(* CODESYS project CANopenExample.project
   Title: CANopen Example

Project tree, tasks and I/O mapping:
  Device : CODESYS Control Win V3 x64, 3S - Smart Software Solutions GmbH, version 3.5.14.0
    application Application
      libraries: Standard, * (System); MemoryUtils, * (3S - Smart Software Solutions GmbH); StringUtils, * (System); CmpLog, * (System); CAA CiA 405, 3.5.14.0 (CAA Technical Workgroup)
      task MainTask (cyclic, interval t#20ms, priority 1) calls CANopenManagerExamples, CANopenLocalDeviceExamples, CANbusExamples
      CANbus Examples/
        program CANbusExamples [ST]
        Change CANbus settings (Reconfigure)/
          program ChangeBaudrate [ST]
          program EnableDisableCANbus [ST]
        Query CANbus/
          function GetCANbus [ST]
      CANopen Master Examples/
        program CANopenManagerExamples [ST]
        CiA405/
          Diagnosis/
            EMCY/
              program ReceiveEMCYFromAllDevicesExample [ST]
              program ReceiveEMCYFromOneDeviceExample [ST]
            State/
              program GetCANopenKernelStateExample [ST]
              program GetStateExample [ST]
          Network management/
            program GetCANopenManagerNodeIDExample [ST]
            program NMT_Example [ST]
          SDO access/
            Block and Segmented/
              program SegmentedAndBlockReadExample [ST]
              program SegmentedAndBlockWriteExample [ST]
            Expedited (<= 4byte)/
              program ExpeditedReadExample [ST]
              program ExpeditedWriteExample [ST]
        Stack API/
          program CANopenManagerAPI [ST]
          program CANopenRemoteDeviceAPI [ST]
          Events/
            function block CANopenManagerEventHandler [ST]: EventCallback
      CANopen Slave Examples/
        program CANopenLocalDeviceExamples [ST]
        Diagnosis/
          function GetLocalDeviceInfoExample [ST]
        Network management/
          program ChangeNodeIDExample [ST]
          program NMTExample [ST]
          data type NMT_Command
        Object Dictionary Access/
          Event Handler/
            function block ObjectDictionaryEventHandler [ST]: OnObjectChanged, OnReadObject, OnWriteObject
            function TO_HEXSTRING [ST]
          Read Object/
            program ReadObjectExample1 [ST]
            program ReadObjectExample2 [ST]
          Traverse object dictionary/
            program CountObjects [ST]
            program GetPDOInfo [ST]
          Write Object/
            program WriteObjectExample1 [ST]
            program WriteObjectExample2 [ST]
      license
    CANbus : CANbus, 3S - Smart Software Solutions GmbH, version 3.5.12.0
        settings: Baudrate = 1000 kbit/s
      CANopen_Manager : CANopen_Manager, 3S - Smart Software Solutions GmbH, version 3.5.10.0
          settings: ConfigVersion = 50659584
        CANopenRemoteDevice : CANopenDeviceExample, 3S - Smart Software Solutions GmbH, order no. 0, version Revision=16#00000004, FileVersion=1.0
            settings: NODEIDSAVED = 1; SDO Timeout = 1000000; EXPERTSETTINGS = FALSE; Heartbeat-Producer Time = 200; PDO 16#1400.COBID = 16#00000201; Process by CANopenManager = TRUE; PDO 16#1800.COBID = 16#00000181; Process by CANopenManager = TRUE; Heartbeat-Consuming1.Heartbeat-Time = 300 ms; DigOutput8.Subindex = 16#01; DigOutput8.Subindex = 16#02; DigOutput8.Subindex = 16#03; DigOutput8.Subindex = 16#04; DigOutput8.Subindex = 16#05; DigOutput8.Subindex = 16#06; DigOutput8.Subindex = 16#07; DigOutput8.Subindex = 16#08; DigInput8.Subindex = 16#01; DigInput8.Subindex = 16#02; DigInput8.Subindex = 16#03; DigInput8.Subindex = 16#04; DigInput8.Subindex = 16#05; DigInput8.Subindex = 16#06; DigInput8.Subindex = 16#07; DigInput8.Subindex = 16#08; SDO List.Set Guardtime.Index = 16#100C; SDO List.Set Guardtime.Subindex = 16#00; SDO List.Set Guardtime.Value = 16#00000000; SDO List.Set Guardtime.Size = 16; SDO List.Set Guardtime.AbortIfError = FALSE; SDO List.Set Guardtime.JumpToLine = FALSE; SDO List.Set Guardtime.Line = 0; SDO List.Set Lifetime.Index = 16#100D; SDO List.Set Lifetime.Subindex = 16#00; SDO List.Set Lifetime.Value = 16#00000000; SDO List.Set Lifetime.Size = 8; SDO List.Set Lifetime.AbortIfError = FALSE; SDO List.Set Lifetime.JumpToLine = FALSE; SDO List.Set Lifetime.Line = 0; SDO List.Disable Emcy CobID.Index = 16#1014;
              SDO List.Disable Emcy CobID.Subindex = 16#00; SDO List.Disable Emcy CobID.Value = 16#80000081; SDO List.Disable Emcy CobID.Size = 32; SDO List.Disable Emcy CobID.AbortIfError = FALSE; SDO List.Disable Emcy CobID.JumpToLine = FALSE; SDO List.Disable Emcy CobID.Line = 0; SDO List.Set Emcy CobID.Index = 16#1014; SDO List.Set Emcy CobID.Subindex = 16#00; SDO List.Set Emcy CobID.Value = 16#00000081; SDO List.Set Emcy CobID.Size = 32; SDO List.Set Emcy CobID.AbortIfError = FALSE; SDO List.Set Emcy CobID.JumpToLine = FALSE; SDO List.Set Emcy CobID.Line = 0; SDO List.Set Heartbeat Consumer.Index = 16#1016; SDO List.Set Heartbeat Consumer.Subindex = 16#01; SDO List.Set Heartbeat Consumer.Value = 16#007F012C; SDO List.Set Heartbeat Consumer.Size = 32; SDO List.Set Heartbeat Consumer.AbortIfError = FALSE; SDO List.Set Heartbeat Consumer.JumpToLine = FALSE; SDO List.Set Heartbeat Consumer.Line = 0; SDO List.Set Heartbeat Producer.Index = 16#1017; SDO List.Set Heartbeat Producer.Subindex = 16#00; SDO List.Set Heartbeat Producer.Value = 16#000000C8; SDO List.Set Heartbeat Producer.Size = 16; SDO List.Set Heartbeat Producer.AbortIfError = FALSE; SDO List.Set Heartbeat Producer.JumpToLine = FALSE; SDO List.Set Heartbeat Producer.Line = 0; SDO List.Disable PDO.Index = 16#1400; SDO List.Disable PDO.Subindex = 16#01; SDO List.Disable PDO.Value = 16#80000201; SDO List.Disable PDO.Size = 32; SDO List.Disable PDO.AbortIfError = FALSE; SDO List.Disable PDO.JumpToLine = FALSE; SDO List.Disable PDO.Line = 0; SDO List.Set transmission type.Index = 16#1400; SDO List.Set transmission type.Subindex = 16#02; SDO List.Set transmission type.Value = 16#FF; SDO List.Set transmission type.Size = 8; SDO List.Set transmission type.AbortIfError = FALSE; SDO List.Set transmission type.JumpToLine = FALSE;
              SDO List.Set transmission type.Line = 0; SDO List.Set and enable COB-ID.Index = 16#1400; SDO List.Set and enable COB-ID.Subindex = 16#01; SDO List.Set and enable COB-ID.Value = 16#00000201; SDO List.Set and enable COB-ID.Size = 32; SDO List.Set and enable COB-ID.AbortIfError = FALSE; SDO List.Set and enable COB-ID.JumpToLine = FALSE; SDO List.Set and enable COB-ID.Line = 0; SDO List.Disable PDO.Index = 16#1800; SDO List.Disable PDO.Subindex = 16#01; SDO List.Disable PDO.Value = 16#80000181; SDO List.Disable PDO.Size = 32; SDO List.Disable PDO.AbortIfError = FALSE; SDO List.Disable PDO.JumpToLine = FALSE; SDO List.Disable PDO.Line = 0; SDO List.Set transmission type.Index = 16#1800; SDO List.Set transmission type.Subindex = 16#02; SDO List.Set transmission type.Value = 16#FF; SDO List.Set transmission type.Size = 8; SDO List.Set transmission type.AbortIfError = FALSE; SDO List.Set transmission type.JumpToLine = FALSE; SDO List.Set transmission type.Line = 0; SDO List.Set inhibit time.Index = 16#1800; SDO List.Set inhibit time.Subindex = 16#03; SDO List.Set inhibit time.Value = 16#0000; SDO List.Set inhibit time.Size = 16; SDO List.Set inhibit time.AbortIfError = FALSE; SDO List.Set inhibit time.JumpToLine = FALSE; SDO List.Set inhibit time.Line = 0; SDO List.Set event time.Index = 16#1800; SDO List.Set event time.Subindex = 16#05; SDO List.Set event time.Value = 16#0000; SDO List.Set event time.Size = 16; SDO List.Set event time.AbortIfError = FALSE; SDO List.Set event time.JumpToLine = FALSE; SDO List.Set event time.Line = 0; SDO List.Set and enable COB-ID.Index = 16#1800; SDO List.Set and enable COB-ID.Subindex = 16#01; SDO List.Set and enable COB-ID.Value = 16#00000181; SDO List.Set and enable COB-ID.Size = 32;
              SDO List.Set and enable COB-ID.AbortIfError = FALSE; SDO List.Set and enable COB-ID.JumpToLine = FALSE; SDO List.Set and enable COB-ID.Line = 0; ConfigVersion = 50659584
            unmapped channels: DigOutput8, DigOutput8, DigOutput8, DigOutput8, DigOutput8, DigOutput8, DigOutput8, DigOutput8, DigInput8, DigInput8, DigInput8, DigInput8, DigInput8, DigInput8, DigInput8, DigInput8
    CANbus_1 : CANbus, 3S - Smart Software Solutions GmbH, version 3.5.12.0
        settings: Baudrate = 1000 kbit/s
      CANopenLocalDevice : CANopen Device, 3S - Smart Software Solutions GmbH, version 3.5.13.0
          settings: Product Name = 'CANopenDeviceExample'; OD_ObjectCount = 16#0015; Objects.Objects = (wIndex := 16#1000, bySubCnt := 16#1); Objects.Objects = (wIndex := 16#1001, bySubCnt := 16#1); Objects.Objects = (wIndex := 16#1003, bySubCnt := 16#04); Objects.Objects = (wIndex := 16#1005, bySubCnt := 16#1); Objects.Objects = (wIndex := 16#1006, bySubCnt := 16#1); Objects.Objects = (wIndex := 16#1008, bySubCnt := 16#1); Objects.Objects = (wIndex := 16#100C, bySubCnt := 16#1); Objects.Objects = (wIndex := 16#100D, bySubCnt := 16#1); Objects.Objects = (wIndex := 16#1014, bySubCnt := 16#1); Objects.Objects = (wIndex := 16#1016, bySubCnt := 16#02); Objects.Objects = (wIndex := 16#1017, bySubCnt := 16#1); Objects.Objects = (wIndex := 16#1018, bySubCnt := 16#04); Objects.Objects = (wIndex := 16#1200, bySubCnt := 16#03); Objects.Objects = (wIndex := 16#1400, bySubCnt := 16#03); Objects.Objects = (wIndex := 16#1600, bySubCnt := 16#09); Objects.Objects = (wIndex := 16#1800, bySubCnt := 16#06); Objects.Objects = (wIndex := 16#1A00, bySubCnt := 16#09); Objects.Objects = (wIndex := 16#3000, bySubCnt := 16#1); Objects.Objects = (wIndex := 16#6000, bySubCnt := 16#09); Objects.Objects = (wIndex := 16#6200, bySubCnt := 16#09); Objects.Objects = (wIndex := 16#6412, bySubCnt := 16#02); SubObjects.SubObjects = (eObjProperties := 16#0001, eDataType := 16#05, udiSize := 16#00000001, xwData := 0, xwDefault := 0, bySubIdx := 16#00); SubObjects.SubObjects = (eObjProperties := 16#0003, eDataType := 16#05, udiSize := 16#00000001, xwData := 0, xwDefault := 0, bySubIdx := 16#00); SubObjects.SubObjects = (eObjProperties := 16#0001, eDataType := 16#07, udiSize := 16#00000004, xwData := 0, xwDefault := 0, bySubIdx := 16#01); SubObjects.SubObjects = (eObjProperties := 16#0001, eDataType := 16#07, udiSize := 16#00000004, xwData := 0, xwDefault := 0, bySubIdx := 16#02); SubObjects.SubObjects = (eObjProperties := 16#0001, eDataType := 16#07, udiSize := 16#00000004, xwData := 0, xwDefault := 0, bySubIdx := 16#03); SubObjects.SubObjects = (eObjProperties := 16#0003, eDataType := 16#07, udiSize := 16#00000004, xwData := 0, xwDefault := 0, bySubIdx := 16#00); SubObjects.SubObjects = (eObjProperties := 16#0001, eDataType := 16#09, udiSize := 20, xwData := 0, xwDefault := 0, bySubIdx := 16#00); SubObjects.SubObjects = (eObjProperties := 16#0003, eDataType := 16#06, udiSize := 16#00000002, xwData := 0, xwDefault := 0, bySubIdx := 16#00); SubObjects.SubObjects = (eObjProperties := 16#0003, eDataType := 16#05, udiSize := 16#00000001, xwData := 0, xwDefault := 0, bySubIdx := 16#00); SubObjects.SubObjects = (eObjProperties := 16#0001, eDataType := 16#05, udiSize := 16#00000001, xwData := 0, xwDefault := 1, bySubIdx := 16#00); SubObjects.SubObjects = (eObjProperties := 16#0003, eDataType := 16#07, udiSize := 16#00000004, xwData := 0, xwDefault := 0, bySubIdx := 16#01); SubObjects.SubObjects = (eObjProperties := 16#0003, eDataType := 16#06, udiSize := 16#00000002, xwData := 0, xwDefault := 0, bySubIdx := 16#00); SubObjects.SubObjects = (eObjProperties := 16#0001, eDataType := 16#05, udiSize := 16#00000001, xwData := 0, xwDefault := 3, bySubIdx := 16#00); SubObjects.SubObjects = (eObjProperties := 16#0001, eDataType := 16#07, udiSize := 16#00000004, xwData := 0, xwDefault := 4, bySubIdx := 16#03); SubObjects.SubObjects = (eObjProperties := 16#0001, eDataType := 16#05, udiSize := 16#00000001, xwData := 0, xwDefault := 2, bySubIdx := 16#00); SubObjects.SubObjects = (eObjProperties := 16#0001, eDataType := 16#05, udiSize := 16#00000001, xwData := 0, xwDefault := 2, bySubIdx := 16#00); SubObjects.SubObjects = (eObjProperties := 16#0001, eDataType := 16#05, udiSize := 16#00000001, xwData := 0, xwDefault := 8, bySubIdx := 16#00);
            SubObjects.SubObjects = (eObjProperties := 16#0001, eDataType := 16#05, udiSize := 16#00000001, xwData := 0, xwDefault := 5, bySubIdx := 16#00); SubObjects.SubObjects = (eObjProperties := 16#0003, eDataType := 16#06, udiSize := 16#00000002, xwData := 0, xwDefault := 0, bySubIdx := 16#03); SubObjects.SubObjects = (eObjProperties := 16#0003, eDataType := 16#05, udiSize := 16#00000001, xwData := 0, xwDefault := 0, bySubIdx := 16#04); SubObjects.SubObjects = (eObjProperties := 16#0003, eDataType := 16#06, udiSize := 16#00000002, xwData := 0, xwDefault := 0, bySubIdx := 16#05); SubObjects.SubObjects = (eObjProperties := 16#0001, eDataType := 16#05, udiSize := 16#00000001, xwData := 0, xwDefault := 8, bySubIdx := 16#00); SubObjects.SubObjects = (eObjProperties := 16#0001, eDataType := 16#05, udiSize := 16#00000001, xwData := 0, xwDefault := 8, bySubIdx := 16#00); SubObjects.SubObjects = (eObjProperties := 16#0001, eDataType := 16#05, udiSize := 16#00000001, xwData := 0, xwDefault := 0, bySubIdx := 16#01); SubObjects.SubObjects = (eObjProperties := 16#0001, eDataType := 16#05, udiSize := 16#00000001, xwData := 0, xwDefault := 0, bySubIdx := 16#02); SubObjects.SubObjects = (eObjProperties := 16#0001, eDataType := 16#05, udiSize := 16#00000001, xwData := 0, xwDefault := 0, bySubIdx := 16#03); SubObjects.SubObjects = (eObjProperties := 16#0001, eDataType := 16#05, udiSize := 16#00000001, xwData := 0, xwDefault := 0, bySubIdx := 16#04); SubObjects.SubObjects = (eObjProperties := 16#0001, eDataType := 16#05, udiSize := 16#00000001, xwData := 0, xwDefault := 0, bySubIdx := 16#05); SubObjects.SubObjects = (eObjProperties := 16#0001, eDataType := 16#05, udiSize := 16#00000001, xwData := 0, xwDefault := 0, bySubIdx := 16#06); SubObjects.SubObjects = (eObjProperties := 16#0001, eDataType := 16#05, udiSize := 16#00000001, xwData := 0, xwDefault := 0, bySubIdx := 16#07); SubObjects.SubObjects = (eObjProperties := 16#0001, eDataType := 16#05, udiSize := 16#00000001, xwData := 0, xwDefault := 0, bySubIdx := 16#08); SubObjects.SubObjects = (eObjProperties := 16#0001, eDataType := 16#05, udiSize := 16#00000001, xwData := 0, xwDefault := 8, bySubIdx := 16#00); SubObjects.SubObjects = (eObjProperties := 16#0003, eDataType := 16#05, udiSize := 16#00000001, xwData := 0, xwDefault := 0, bySubIdx := 16#01); SubObjects.SubObjects = (eObjProperties := 16#0003, eDataType := 16#05, udiSize := 16#00000001, xwData := 0, xwDefault := 0, bySubIdx := 16#02); SubObjects.SubObjects = (eObjProperties := 16#0003, eDataType := 16#05, udiSize := 16#00000001, xwData := 0, xwDefault := 0, bySubIdx := 16#03); SubObjects.SubObjects = (eObjProperties := 16#0003, eDataType := 16#05, udiSize := 16#00000001, xwData := 0, xwDefault := 0, bySubIdx := 16#04); SubObjects.SubObjects = (eObjProperties := 16#0003, eDataType := 16#05, udiSize := 16#00000001, xwData := 0, xwDefault := 0, bySubIdx := 16#05); SubObjects.SubObjects = (eObjProperties := 16#0003, eDataType := 16#05, udiSize := 16#00000001, xwData := 0, xwDefault := 0, bySubIdx := 16#06); SubObjects.SubObjects = (eObjProperties := 16#0003, eDataType := 16#05, udiSize := 16#00000001, xwData := 0, xwDefault := 0, bySubIdx := 16#07); SubObjects.SubObjects = (eObjProperties := 16#0003, eDataType := 16#05, udiSize := 16#00000001, xwData := 0, xwDefault := 0, bySubIdx := 16#08); SubObjects.SubObjects = (eObjProperties := 16#0001, eDataType := 16#05, udiSize := 16#00000001, xwData := 0, xwDefault := 1, bySubIdx := 16#00); SubObjects.SubObjects = (eObjProperties := 16#0003, eDataType := 16#04, udiSize := 16#00000004, xwData := 0, xwDefault := 0, bySubIdx := 16#01); ObjectsOfflineInfo.Predefined Error Field.Index = 16#00001003; ObjectsOfflineInfo.Predefined Error Field.ObjectOwner = 16#00; ObjectsOfflineInfo.Predefined Error Field.ObjectType = 16#00000008; ObjectsOfflineInfo.Predefined Error Field.ObjectFlags = 16#00000000; ObjectsOfflineInfo.Consumer Heartbeat Time.Index = 16#00001016; ObjectsOfflineInfo.Consumer Heartbeat Time.ObjectOwner = 16#00; ObjectsOfflineInfo.Consumer Heartbeat Time.ObjectType = 16#00000008; ObjectsOfflineInfo.Consumer Heartbeat Time.ObjectFlags = 16#00000000; ObjectsOfflineInfo.Identity Object.Index = 16#00001018; ObjectsOfflineInfo.Identity Object.ObjectOwner = 16#00; ObjectsOfflineInfo.Identity Object.ObjectType = 16#00000009; ObjectsOfflineInfo.Identity Object.ObjectFlags = 16#00000000; ObjectsOfflineInfo.ServerSdoParameter.Index = 16#00001200; ObjectsOfflineInfo.ServerSdoParameter.ObjectOwner = 16#00; ObjectsOfflineInfo.ServerSdoParameter.ObjectType = 16#00000009;
            ObjectsOfflineInfo.ServerSdoParameter.ObjectFlags = 16#00000000; ObjectsOfflineInfo.RPDO communication parameter.Index = 16#00001400; ObjectsOfflineInfo.RPDO communication parameter.ObjectOwner = 16#03; ObjectsOfflineInfo.RPDO communication parameter.ObjectType = 16#00000009; ObjectsOfflineInfo.RPDO communication parameter.ObjectFlags = 16#00000000; ObjectsOfflineInfo.RPDO mapping parameter.Index = 16#00001600; ObjectsOfflineInfo.RPDO mapping parameter.ObjectOwner = 16#03; ObjectsOfflineInfo.RPDO mapping parameter.ObjectType = 16#00000009; ObjectsOfflineInfo.RPDO mapping parameter.ObjectFlags = 16#00000000; ObjectsOfflineInfo.TPDO communication parameter.Index = 16#00001800; ObjectsOfflineInfo.TPDO communication parameter.ObjectOwner = 16#03; ObjectsOfflineInfo.TPDO communication parameter.ObjectType = 16#00000009; ObjectsOfflineInfo.TPDO communication parameter.ObjectFlags = 16#00000000; ObjectsOfflineInfo.TPDO mapping parameter.Index = 16#00001A00; ObjectsOfflineInfo.TPDO mapping parameter.ObjectOwner = 16#03; ObjectsOfflineInfo.TPDO mapping parameter.ObjectType = 16#00000009; ObjectsOfflineInfo.TPDO mapping parameter.ObjectFlags = 16#00000000; ObjectsOfflineInfo.Read Input 8 Bit.Index = 16#00006000; ObjectsOfflineInfo.Read Input 8 Bit.ObjectOwner = 16#03; ObjectsOfflineInfo.Read Input 8 Bit.ObjectType = 16#00000008; ObjectsOfflineInfo.Read Input 8 Bit.ObjectFlags = 16#00000000; ObjectsOfflineInfo.Write Output 8 Bit.Index = 16#00006200; ObjectsOfflineInfo.Write Output 8 Bit.ObjectOwner = 16#03; ObjectsOfflineInfo.Write Output 8 Bit.ObjectType = 16#00000008; ObjectsOfflineInfo.Write Output 8 Bit.ObjectFlags = 16#00000000; ObjectsOfflineInfo.Write Analogue Output 32 Bit.Index = 16#00006412; ObjectsOfflineInfo.Write Analogue Output 32 Bit.ObjectOwner = 16#03; ObjectsOfflineInfo.Write Analogue Output 32 Bit.ObjectType = 16#00000008; ObjectsOfflineInfo.Write Analogue Output 32 Bit.ObjectFlags = 16#00000000; SubObjectsOfflineInfo.Device Type.Index = 16#00001000; SubObjectsOfflineInfo.Device Type.SubIndex = 16#00; SubObjectsOfflineInfo.Device Type.PDOMapping = FALSE; SubObjectsOfflineInfo.Device Type.ObjectOwner = 16#00; SubObjectsOfflineInfo.Device Type.ObjectType = 16#00000007; SubObjectsOfflineInfo.Device Type.MinValue = ''; SubObjectsOfflineInfo.Device Type.MaxValue = ''; SubObjectsOfflineInfo.Device Type.AccessType = 'ro'; SubObjectsOfflineInfo.Device Type.IEC Variable = ''; SubObjectsOfflineInfo.Device Type.DefaultValue = '0x191'; SubObjectsOfflineInfo.Device Type.ObjectFlags = 16#00000000;
            SubObjectsOfflineInfo.Error Register.Index = 16#00001001; SubObjectsOfflineInfo.Error Register.SubIndex = 16#00; SubObjectsOfflineInfo.Error Register.PDOMapping = FALSE; SubObjectsOfflineInfo.Error Register.ObjectOwner = 16#00; SubObjectsOfflineInfo.Error Register.ObjectType = 16#00000007; SubObjectsOfflineInfo.Error Register.MinValue = ''; SubObjectsOfflineInfo.Error Register.MaxValue = ''; SubObjectsOfflineInfo.Error Register.AccessType = 'ro'; SubObjectsOfflineInfo.Error Register.IEC Variable = ''; SubObjectsOfflineInfo.Error Register.DefaultValue = '0x0'; SubObjectsOfflineInfo.Error Register.ObjectFlags = 16#00000000; SubObjectsOfflineInfo.Number of Errors.Index = 16#00001003; SubObjectsOfflineInfo.Number of Errors.SubIndex = 16#00; SubObjectsOfflineInfo.Number of Errors.PDOMapping = FALSE; SubObjectsOfflineInfo.Number of Errors.ObjectOwner = 16#00; SubObjectsOfflineInfo.Number of Errors.ObjectType = 16#00000007; SubObjectsOfflineInfo.Number of Errors.MinValue = ''; SubObjectsOfflineInfo.Number of Errors.MaxValue = ''; SubObjectsOfflineInfo.Number of Errors.AccessType = 'rw'; SubObjectsOfflineInfo.Number of Errors.IEC Variable = ''; SubObjectsOfflineInfo.Number of Errors.DefaultValue = '0'; SubObjectsOfflineInfo.Number of Errors.ObjectFlags = 16#00000000; SubObjectsOfflineInfo.Standard Error Field.Index = 16#00001003; SubObjectsOfflineInfo.Standard Error Field.SubIndex = 16#01; SubObjectsOfflineInfo.Standard Error Field.PDOMapping = FALSE; SubObjectsOfflineInfo.Standard Error Field.ObjectOwner = 16#00; SubObjectsOfflineInfo.Standard Error Field.ObjectType = 16#00000007; SubObjectsOfflineInfo.Standard Error Field.MinValue = ''; SubObjectsOfflineInfo.Standard Error Field.MaxValue = ''; SubObjectsOfflineInfo.Standard Error Field.AccessType = 'ro'; SubObjectsOfflineInfo.Standard Error Field.IEC Variable = ''; SubObjectsOfflineInfo.Standard Error Field.DefaultValue = ''; SubObjectsOfflineInfo.Standard Error Field.ObjectFlags = 16#00000000; SubObjectsOfflineInfo.Standard Error Field 2.Index = 16#00001003; SubObjectsOfflineInfo.Standard Error Field 2.SubIndex = 16#02; SubObjectsOfflineInfo.Standard Error Field 2.PDOMapping = FALSE; SubObjectsOfflineInfo.Standard Error Field 2.ObjectOwner = 16#00; SubObjectsOfflineInfo.Standard Error Field 2.ObjectType = 16#00000007; SubObjectsOfflineInfo.Standard Error Field 2.MinValue = ''; SubObjectsOfflineInfo.Standard Error Field 2.MaxValue = '';
            SubObjectsOfflineInfo.Standard Error Field 2.AccessType = 'ro'; SubObjectsOfflineInfo.Standard Error Field 2.IEC Variable = ''; SubObjectsOfflineInfo.Standard Error Field 2.DefaultValue = ''; SubObjectsOfflineInfo.Standard Error Field 2.ObjectFlags = 16#00000000; SubObjectsOfflineInfo.Standard Error Field 3.Index = 16#00001003; SubObjectsOfflineInfo.Standard Error Field 3.SubIndex = 16#03; SubObjectsOfflineInfo.Standard Error Field 3.PDOMapping = FALSE; SubObjectsOfflineInfo.Standard Error Field 3.ObjectOwner = 16#00; SubObjectsOfflineInfo.Standard Error Field 3.ObjectType = 16#00000007; SubObjectsOfflineInfo.Standard Error Field 3.MinValue = ''; SubObjectsOfflineInfo.Standard Error Field 3.MaxValue = ''; SubObjectsOfflineInfo.Standard Error Field 3.AccessType = 'ro'; SubObjectsOfflineInfo.Standard Error Field 3.IEC Variable = ''; SubObjectsOfflineInfo.Standard Error Field 3.DefaultValue = ''; SubObjectsOfflineInfo.Standard Error Field 3.ObjectFlags = 16#00000000; SubObjectsOfflineInfo.Sync COB-ID.Index = 16#00001005; SubObjectsOfflineInfo.Sync COB-ID.SubIndex = 16#00; SubObjectsOfflineInfo.Sync COB-ID.PDOMapping = FALSE; SubObjectsOfflineInfo.Sync COB-ID.ObjectOwner = 16#00; SubObjectsOfflineInfo.Sync COB-ID.ObjectType = 16#00000007; SubObjectsOfflineInfo.Sync COB-ID.MinValue = ''; SubObjectsOfflineInfo.Sync COB-ID.MaxValue = ''; SubObjectsOfflineInfo.Sync COB-ID.AccessType = 'rw'; SubObjectsOfflineInfo.Sync COB-ID.IEC Variable = ''; SubObjectsOfflineInfo.Sync COB-ID.DefaultValue = '0x80'; SubObjectsOfflineInfo.Sync COB-ID.ObjectFlags = 16#00000000; SubObjectsOfflineInfo.Communication Cycle Period.Index = 16#00001006; SubObjectsOfflineInfo.Communication Cycle Period.SubIndex = 16#00; SubObjectsOfflineInfo.Communication Cycle Period.PDOMapping = FALSE; SubObjectsOfflineInfo.Communication Cycle Period.ObjectOwner = 16#00; SubObjectsOfflineInfo.Communication Cycle Period.ObjectType = 16#00000007; SubObjectsOfflineInfo.Communication Cycle Period.MinValue = ''; SubObjectsOfflineInfo.Communication Cycle Period.MaxValue = ''; SubObjectsOfflineInfo.Communication Cycle Period.AccessType = 'rw'; SubObjectsOfflineInfo.Communication Cycle Period.IEC Variable = ''; SubObjectsOfflineInfo.Communication Cycle Period.DefaultValue = '0x0'; SubObjectsOfflineInfo.Communication Cycle Period.ObjectFlags = 16#00000000; SubObjectsOfflineInfo.Manufacturer device name.Index = 16#00001008; SubObjectsOfflineInfo.Manufacturer device name.SubIndex = 16#00; SubObjectsOfflineInfo.Manufacturer device name.PDOMapping = FALSE;
            SubObjectsOfflineInfo.Manufacturer device name.ObjectOwner = 16#03; SubObjectsOfflineInfo.Manufacturer device name.ObjectType = 16#00000007; SubObjectsOfflineInfo.Manufacturer device name.MinValue = ''; SubObjectsOfflineInfo.Manufacturer device name.MaxValue = ''; SubObjectsOfflineInfo.Manufacturer device name.AccessType = 'const'; SubObjectsOfflineInfo.Manufacturer device name.IEC Variable = ''; SubObjectsOfflineInfo.Manufacturer device name.DefaultValue = 'CANopenDeviceExample'; SubObjectsOfflineInfo.Manufacturer device name.ObjectFlags = 16#00000000; SubObjectsOfflineInfo.Guard Time.Index = 16#0000100C; SubObjectsOfflineInfo.Guard Time.SubIndex = 16#00; SubObjectsOfflineInfo.Guard Time.PDOMapping = FALSE; SubObjectsOfflineInfo.Guard Time.ObjectOwner = 16#00; SubObjectsOfflineInfo.Guard Time.ObjectType = 16#00000007; SubObjectsOfflineInfo.Guard Time.MinValue = ''; SubObjectsOfflineInfo.Guard Time.MaxValue = ''; SubObjectsOfflineInfo.Guard Time.AccessType = 'rw'; SubObjectsOfflineInfo.Guard Time.IEC Variable = ''; SubObjectsOfflineInfo.Guard Time.DefaultValue = '0x0'; SubObjectsOfflineInfo.Guard Time.ObjectFlags = 16#00000000; SubObjectsOfflineInfo.Life Time Factor.Index = 16#0000100D; SubObjectsOfflineInfo.Life Time Factor.SubIndex = 16#00; SubObjectsOfflineInfo.Life Time Factor.PDOMapping = FALSE; SubObjectsOfflineInfo.Life Time Factor.ObjectOwner = 16#00; SubObjectsOfflineInfo.Life Time Factor.ObjectType = 16#00000007; SubObjectsOfflineInfo.Life Time Factor.MinValue = ''; SubObjectsOfflineInfo.Life Time Factor.MaxValue = ''; SubObjectsOfflineInfo.Life Time Factor.AccessType = 'rw'; SubObjectsOfflineInfo.Life Time Factor.IEC Variable = ''; SubObjectsOfflineInfo.Life Time Factor.DefaultValue = '0'; SubObjectsOfflineInfo.Life Time Factor.ObjectFlags = 16#00000000; SubObjectsOfflineInfo.COB-ID EMCY.Index = 16#00001014; SubObjectsOfflineInfo.COB-ID EMCY.SubIndex = 16#00; SubObjectsOfflineInfo.COB-ID EMCY.PDOMapping = FALSE; SubObjectsOfflineInfo.COB-ID EMCY.ObjectOwner = 16#00; SubObjectsOfflineInfo.COB-ID EMCY.ObjectType = 16#00000007; SubObjectsOfflineInfo.COB-ID EMCY.MinValue = ''; SubObjectsOfflineInfo.COB-ID EMCY.MaxValue = ''; SubObjectsOfflineInfo.COB-ID EMCY.AccessType = 'rw'; SubObjectsOfflineInfo.COB-ID EMCY.IEC Variable = ''; SubObjectsOfflineInfo.COB-ID EMCY.DefaultValue = '$$NODEID+0x80';
            SubObjectsOfflineInfo.COB-ID EMCY.ObjectFlags = 16#00000000; SubObjectsOfflineInfo.Number of Entries.Index = 16#00001016; SubObjectsOfflineInfo.Number of Entries.SubIndex = 16#00; SubObjectsOfflineInfo.Number of Entries.PDOMapping = FALSE; SubObjectsOfflineInfo.Number of Entries.ObjectOwner = 16#00; SubObjectsOfflineInfo.Number of Entries.ObjectType = 16#00000007; SubObjectsOfflineInfo.Number of Entries.MinValue = ''; SubObjectsOfflineInfo.Number of Entries.MaxValue = ''; SubObjectsOfflineInfo.Number of Entries.AccessType = 'ro'; SubObjectsOfflineInfo.Number of Entries.IEC Variable = ''; SubObjectsOfflineInfo.Number of Entries.DefaultValue = '0x1'; SubObjectsOfflineInfo.Number of Entries.ObjectFlags = 16#00000000; SubObjectsOfflineInfo.Consumer Heartbeat Time.Index = 16#00001016; SubObjectsOfflineInfo.Consumer Heartbeat Time.SubIndex = 16#01; SubObjectsOfflineInfo.Consumer Heartbeat Time.PDOMapping = FALSE; SubObjectsOfflineInfo.Consumer Heartbeat Time.ObjectOwner = 16#00; SubObjectsOfflineInfo.Consumer Heartbeat Time.ObjectType = 16#00000007; SubObjectsOfflineInfo.Consumer Heartbeat Time.MinValue = ''; SubObjectsOfflineInfo.Consumer Heartbeat Time.MaxValue = ''; SubObjectsOfflineInfo.Consumer Heartbeat Time.AccessType = 'rw'; SubObjectsOfflineInfo.Consumer Heartbeat Time.IEC Variable = ''; SubObjectsOfflineInfo.Consumer Heartbeat Time.DefaultValue = '0x0'; SubObjectsOfflineInfo.Consumer Heartbeat Time.ObjectFlags = 16#00000000; SubObjectsOfflineInfo.Producer Heartbeat Time.Index = 16#00001017; SubObjectsOfflineInfo.Producer Heartbeat Time.SubIndex = 16#00; SubObjectsOfflineInfo.Producer Heartbeat Time.PDOMapping = FALSE; SubObjectsOfflineInfo.Producer Heartbeat Time.ObjectOwner = 16#00; SubObjectsOfflineInfo.Producer Heartbeat Time.ObjectType = 16#00000007; SubObjectsOfflineInfo.Producer Heartbeat Time.MinValue = ''; SubObjectsOfflineInfo.Producer Heartbeat Time.MaxValue = ''; SubObjectsOfflineInfo.Producer Heartbeat Time.AccessType = 'rw'; SubObjectsOfflineInfo.Producer Heartbeat Time.IEC Variable = ''; SubObjectsOfflineInfo.Producer Heartbeat Time.DefaultValue = '0x0'; SubObjectsOfflineInfo.Producer Heartbeat Time.ObjectFlags = 16#00000000; SubObjectsOfflineInfo.Number of Entries.Index = 16#00001018; SubObjectsOfflineInfo.Number of Entries.SubIndex = 16#00; SubObjectsOfflineInfo.Number of Entries.PDOMapping = FALSE; SubObjectsOfflineInfo.Number of Entries.ObjectOwner = 16#00; SubObjectsOfflineInfo.Number of Entries.ObjectType = 16#00000007; SubObjectsOfflineInfo.Number of Entries.MinValue = '0x1';
            SubObjectsOfflineInfo.Number of Entries.MaxValue = '0x3'; SubObjectsOfflineInfo.Number of Entries.AccessType = 'ro'; SubObjectsOfflineInfo.Number of Entries.IEC Variable = ''; SubObjectsOfflineInfo.Number of Entries.DefaultValue = '3'; SubObjectsOfflineInfo.Number of Entries.ObjectFlags = 16#00000000; SubObjectsOfflineInfo.Vendor Id.Index = 16#00001018; SubObjectsOfflineInfo.Vendor Id.SubIndex = 16#01; SubObjectsOfflineInfo.Vendor Id.PDOMapping = FALSE; SubObjectsOfflineInfo.Vendor Id.ObjectOwner = 16#00; SubObjectsOfflineInfo.Vendor Id.ObjectType = 16#00000007; SubObjectsOfflineInfo.Vendor Id.MinValue = ''; SubObjectsOfflineInfo.Vendor Id.MaxValue = ''; SubObjectsOfflineInfo.Vendor Id.AccessType = 'ro'; SubObjectsOfflineInfo.Vendor Id.IEC Variable = ''; SubObjectsOfflineInfo.Vendor Id.DefaultValue = '801'; SubObjectsOfflineInfo.Vendor Id.ObjectFlags = 16#00000000; SubObjectsOfflineInfo.Product Code.Index = 16#00001018; SubObjectsOfflineInfo.Product Code.SubIndex = 16#02; SubObjectsOfflineInfo.Product Code.PDOMapping = FALSE; SubObjectsOfflineInfo.Product Code.ObjectOwner = 16#00; SubObjectsOfflineInfo.Product Code.ObjectType = 16#00000007; SubObjectsOfflineInfo.Product Code.MinValue = ''; SubObjectsOfflineInfo.Product Code.MaxValue = ''; SubObjectsOfflineInfo.Product Code.AccessType = 'ro'; SubObjectsOfflineInfo.Product Code.IEC Variable = ''; SubObjectsOfflineInfo.Product Code.DefaultValue = '30'; SubObjectsOfflineInfo.Product Code.ObjectFlags = 16#00000000; SubObjectsOfflineInfo.Revision Number.Index = 16#00001018; SubObjectsOfflineInfo.Revision Number.SubIndex = 16#03; SubObjectsOfflineInfo.Revision Number.PDOMapping = FALSE; SubObjectsOfflineInfo.Revision Number.ObjectOwner = 16#00; SubObjectsOfflineInfo.Revision Number.ObjectType = 16#00000007; SubObjectsOfflineInfo.Revision Number.MinValue = ''; SubObjectsOfflineInfo.Revision Number.MaxValue = ''; SubObjectsOfflineInfo.Revision Number.AccessType = 'ro'; SubObjectsOfflineInfo.Revision Number.IEC Variable = ''; SubObjectsOfflineInfo.Revision Number.DefaultValue = '4'; SubObjectsOfflineInfo.Revision Number.ObjectFlags = 16#00000000; SubObjectsOfflineInfo.Number of Entries.Index = 16#00001200; SubObjectsOfflineInfo.Number of Entries.SubIndex = 16#00;
            SubObjectsOfflineInfo.Number of Entries.PDOMapping = FALSE; SubObjectsOfflineInfo.Number of Entries.ObjectOwner = 16#00; SubObjectsOfflineInfo.Number of Entries.ObjectType = 16#00000007; SubObjectsOfflineInfo.Number of Entries.MinValue = '0x2'; SubObjectsOfflineInfo.Number of Entries.MaxValue = '0x2'; SubObjectsOfflineInfo.Number of Entries.AccessType = 'ro'; SubObjectsOfflineInfo.Number of Entries.IEC Variable = ''; SubObjectsOfflineInfo.Number of Entries.DefaultValue = '0x2'; SubObjectsOfflineInfo.Number of Entries.ObjectFlags = 16#00000000; SubObjectsOfflineInfo.COB-ID Client->Server.Index = 16#00001200; SubObjectsOfflineInfo.COB-ID Client->Server.SubIndex = 16#01; SubObjectsOfflineInfo.COB-ID Client->Server.PDOMapping = FALSE; SubObjectsOfflineInfo.COB-ID Client->Server.ObjectOwner = 16#00; SubObjectsOfflineInfo.COB-ID Client->Server.ObjectType = 16#00000007; SubObjectsOfflineInfo.COB-ID Client->Server.MinValue = ''; SubObjectsOfflineInfo.COB-ID Client->Server.MaxValue = ''; SubObjectsOfflineInfo.COB-ID Client->Server.AccessType = 'ro'; SubObjectsOfflineInfo.COB-ID Client->Server.IEC Variable = ''; SubObjectsOfflineInfo.COB-ID Client->Server.DefaultValue = '$$NodeId+0x600'; SubObjectsOfflineInfo.COB-ID Client->Server.ObjectFlags = 16#00000000; SubObjectsOfflineInfo.COB-ID Server->Client.Index = 16#00001200; SubObjectsOfflineInfo.COB-ID Server->Client.SubIndex = 16#02; SubObjectsOfflineInfo.COB-ID Server->Client.PDOMapping = FALSE; SubObjectsOfflineInfo.COB-ID Server->Client.ObjectOwner = 16#00; SubObjectsOfflineInfo.COB-ID Server->Client.ObjectType = 16#00000007; SubObjectsOfflineInfo.COB-ID Server->Client.MinValue = ''; SubObjectsOfflineInfo.COB-ID Server->Client.MaxValue = ''; SubObjectsOfflineInfo.COB-ID Server->Client.AccessType = 'ro'; SubObjectsOfflineInfo.COB-ID Server->Client.IEC Variable = ''; SubObjectsOfflineInfo.COB-ID Server->Client.DefaultValue = '$$NodeId+0x580'; SubObjectsOfflineInfo.COB-ID Server->Client.ObjectFlags = 16#00000000; SubObjectsOfflineInfo.Highest sub-index supported.Index = 16#00001400; SubObjectsOfflineInfo.Highest sub-index supported.SubIndex = 16#00; SubObjectsOfflineInfo.Highest sub-index supported.PDOMapping = FALSE; SubObjectsOfflineInfo.Highest sub-index supported.ObjectOwner = 16#03; SubObjectsOfflineInfo.Highest sub-index supported.ObjectType = 16#00000007; SubObjectsOfflineInfo.Highest sub-index supported.MinValue = '0x02'; SubObjectsOfflineInfo.Highest sub-index supported.MaxValue = '0x05'; SubObjectsOfflineInfo.Highest sub-index supported.AccessType = 'const'; SubObjectsOfflineInfo.Highest sub-index supported.IEC Variable = '';
            SubObjectsOfflineInfo.Highest sub-index supported.DefaultValue = '0x2'; SubObjectsOfflineInfo.Highest sub-index supported.ObjectFlags = 16#00000000; SubObjectsOfflineInfo.COB-ID used by RPDO.Index = 16#00001400; SubObjectsOfflineInfo.COB-ID used by RPDO.SubIndex = 16#01; SubObjectsOfflineInfo.COB-ID used by RPDO.PDOMapping = FALSE; SubObjectsOfflineInfo.COB-ID used by RPDO.ObjectOwner = 16#03; SubObjectsOfflineInfo.COB-ID used by RPDO.ObjectType = 16#00000007; SubObjectsOfflineInfo.COB-ID used by RPDO.MinValue = '0x00000080'; SubObjectsOfflineInfo.COB-ID used by RPDO.MaxValue = '0xFFFFFFFF'; SubObjectsOfflineInfo.COB-ID used by RPDO.AccessType = 'rw'; SubObjectsOfflineInfo.COB-ID used by RPDO.IEC Variable = ''; SubObjectsOfflineInfo.COB-ID used by RPDO.DefaultValue = '$$NODEID+0x200'; SubObjectsOfflineInfo.COB-ID used by RPDO.ObjectFlags = 16#00000000; SubObjectsOfflineInfo.Transmission Type.Index = 16#00001400; SubObjectsOfflineInfo.Transmission Type.SubIndex = 16#02; SubObjectsOfflineInfo.Transmission Type.PDOMapping = FALSE; SubObjectsOfflineInfo.Transmission Type.ObjectOwner = 16#03; SubObjectsOfflineInfo.Transmission Type.ObjectType = 16#00000007; SubObjectsOfflineInfo.Transmission Type.MinValue = ''; SubObjectsOfflineInfo.Transmission Type.MaxValue = ''; SubObjectsOfflineInfo.Transmission Type.AccessType = 'rw'; SubObjectsOfflineInfo.Transmission Type.IEC Variable = ''; SubObjectsOfflineInfo.Transmission Type.DefaultValue = '0xFF'; SubObjectsOfflineInfo.Transmission Type.ObjectFlags = 16#00000000; SubObjectsOfflineInfo.Number of mapped application objects in PDO.Index = 16#00001600; SubObjectsOfflineInfo.Number of mapped application objects in PDO.SubIndex = 16#00; SubObjectsOfflineInfo.Number of mapped application objects in PDO.PDOMapping = FALSE; SubObjectsOfflineInfo.Number of mapped application objects in PDO.ObjectOwner = 16#03; SubObjectsOfflineInfo.Number of mapped application objects in PDO.ObjectType = 16#00000007; SubObjectsOfflineInfo.Number of mapped application objects in PDO.MinValue = '0x00'; SubObjectsOfflineInfo.Number of mapped application objects in PDO.MaxValue = '0xFF'; SubObjectsOfflineInfo.Number of mapped application objects in PDO.AccessType = 'const'; SubObjectsOfflineInfo.Number of mapped application objects in PDO.IEC Variable = ''; SubObjectsOfflineInfo.Number of mapped application objects in PDO.DefaultValue = '0x08'; SubObjectsOfflineInfo.Number of mapped application objects in PDO.ObjectFlags = 16#00000000; SubObjectsOfflineInfo.PDO Mapping Entry.Index = 16#00001600; SubObjectsOfflineInfo.PDO Mapping Entry.SubIndex = 16#01; SubObjectsOfflineInfo.PDO Mapping Entry.PDOMapping = FALSE; SubObjectsOfflineInfo.PDO Mapping Entry.ObjectOwner = 16#03; SubObjectsOfflineInfo.PDO Mapping Entry.ObjectType = 16#00000007;
            SubObjectsOfflineInfo.PDO Mapping Entry.MinValue = ''; SubObjectsOfflineInfo.PDO Mapping Entry.MaxValue = ''; SubObjectsOfflineInfo.PDO Mapping Entry.AccessType = 'const'; SubObjectsOfflineInfo.PDO Mapping Entry.IEC Variable = ''; SubObjectsOfflineInfo.PDO Mapping Entry.DefaultValue = '0x62000108'; SubObjectsOfflineInfo.PDO Mapping Entry.ObjectFlags = 16#00000000; SubObjectsOfflineInfo.PDO Mapping Entry.Index = 16#00001600; SubObjectsOfflineInfo.PDO Mapping Entry.SubIndex = 16#02; SubObjectsOfflineInfo.PDO Mapping Entry.PDOMapping = FALSE; SubObjectsOfflineInfo.PDO Mapping Entry.ObjectOwner = 16#03; SubObjectsOfflineInfo.PDO Mapping Entry.ObjectType = 16#00000007; SubObjectsOfflineInfo.PDO Mapping Entry.MinValue = ''; SubObjectsOfflineInfo.PDO Mapping Entry.MaxValue = ''; SubObjectsOfflineInfo.PDO Mapping Entry.AccessType = 'const'; SubObjectsOfflineInfo.PDO Mapping Entry.IEC Variable = ''; SubObjectsOfflineInfo.PDO Mapping Entry.DefaultValue = '0x62000208'; SubObjectsOfflineInfo.PDO Mapping Entry.ObjectFlags = 16#00000000; SubObjectsOfflineInfo.PDO Mapping Entry.Index = 16#00001600; SubObjectsOfflineInfo.PDO Mapping Entry.SubIndex = 16#03; SubObjectsOfflineInfo.PDO Mapping Entry.PDOMapping = FALSE; SubObjectsOfflineInfo.PDO Mapping Entry.ObjectOwner = 16#03; SubObjectsOfflineInfo.PDO Mapping Entry.ObjectType = 16#00000007; SubObjectsOfflineInfo.PDO Mapping Entry.MinValue = ''; SubObjectsOfflineInfo.PDO Mapping Entry.MaxValue = ''; SubObjectsOfflineInfo.PDO Mapping Entry.AccessType = 'const'; SubObjectsOfflineInfo.PDO Mapping Entry.IEC Variable = ''; SubObjectsOfflineInfo.PDO Mapping Entry.DefaultValue = '0x62000308'; SubObjectsOfflineInfo.PDO Mapping Entry.ObjectFlags = 16#00000000; SubObjectsOfflineInfo.PDO Mapping Entry.Index = 16#00001600; SubObjectsOfflineInfo.PDO Mapping Entry.SubIndex = 16#04; SubObjectsOfflineInfo.PDO Mapping Entry.PDOMapping = FALSE; SubObjectsOfflineInfo.PDO Mapping Entry.ObjectOwner = 16#03; SubObjectsOfflineInfo.PDO Mapping Entry.ObjectType = 16#00000007; SubObjectsOfflineInfo.PDO Mapping Entry.MinValue = ''; SubObjectsOfflineInfo.PDO Mapping Entry.MaxValue = ''; SubObjectsOfflineInfo.PDO Mapping Entry.AccessType = 'const'; SubObjectsOfflineInfo.PDO Mapping Entry.IEC Variable = ''; SubObjectsOfflineInfo.PDO Mapping Entry.DefaultValue = '0x62000408'; SubObjectsOfflineInfo.PDO Mapping Entry.ObjectFlags = 16#00000000; SubObjectsOfflineInfo.PDO Mapping Entry.Index = 16#00001600;
            SubObjectsOfflineInfo.PDO Mapping Entry.SubIndex = 16#05; SubObjectsOfflineInfo.PDO Mapping Entry.PDOMapping = FALSE; SubObjectsOfflineInfo.PDO Mapping Entry.ObjectOwner = 16#03; SubObjectsOfflineInfo.PDO Mapping Entry.ObjectType = 16#00000007; SubObjectsOfflineInfo.PDO Mapping Entry.MinValue = ''; SubObjectsOfflineInfo.PDO Mapping Entry.MaxValue = ''; SubObjectsOfflineInfo.PDO Mapping Entry.AccessType = 'const'; SubObjectsOfflineInfo.PDO Mapping Entry.IEC Variable = ''; SubObjectsOfflineInfo.PDO Mapping Entry.DefaultValue = '0x62000508'; SubObjectsOfflineInfo.PDO Mapping Entry.ObjectFlags = 16#00000000; SubObjectsOfflineInfo.PDO Mapping Entry.Index = 16#00001600; SubObjectsOfflineInfo.PDO Mapping Entry.SubIndex = 16#06; SubObjectsOfflineInfo.PDO Mapping Entry.PDOMapping = FALSE; SubObjectsOfflineInfo.PDO Mapping Entry.ObjectOwner = 16#03; SubObjectsOfflineInfo.PDO Mapping Entry.ObjectType = 16#00000007; SubObjectsOfflineInfo.PDO Mapping Entry.MinValue = ''; SubObjectsOfflineInfo.PDO Mapping Entry.MaxValue = ''; SubObjectsOfflineInfo.PDO Mapping Entry.AccessType = 'const'; SubObjectsOfflineInfo.PDO Mapping Entry.IEC Variable = ''; SubObjectsOfflineInfo.PDO Mapping Entry.DefaultValue = '0x62000608'; SubObjectsOfflineInfo.PDO Mapping Entry.ObjectFlags = 16#00000000; SubObjectsOfflineInfo.PDO Mapping Entry.Index = 16#00001600; SubObjectsOfflineInfo.PDO Mapping Entry.SubIndex = 16#07; SubObjectsOfflineInfo.PDO Mapping Entry.PDOMapping = FALSE; SubObjectsOfflineInfo.PDO Mapping Entry.ObjectOwner = 16#03; SubObjectsOfflineInfo.PDO Mapping Entry.ObjectType = 16#00000007; SubObjectsOfflineInfo.PDO Mapping Entry.MinValue = ''; SubObjectsOfflineInfo.PDO Mapping Entry.MaxValue = ''; SubObjectsOfflineInfo.PDO Mapping Entry.AccessType = 'const'; SubObjectsOfflineInfo.PDO Mapping Entry.IEC Variable = ''; SubObjectsOfflineInfo.PDO Mapping Entry.DefaultValue = '0x62000708'; SubObjectsOfflineInfo.PDO Mapping Entry.ObjectFlags = 16#00000000; SubObjectsOfflineInfo.PDO Mapping Entry.Index = 16#00001600; SubObjectsOfflineInfo.PDO Mapping Entry.SubIndex = 16#08; SubObjectsOfflineInfo.PDO Mapping Entry.PDOMapping = FALSE; SubObjectsOfflineInfo.PDO Mapping Entry.ObjectOwner = 16#03; SubObjectsOfflineInfo.PDO Mapping Entry.ObjectType = 16#00000007; SubObjectsOfflineInfo.PDO Mapping Entry.MinValue = ''; SubObjectsOfflineInfo.PDO Mapping Entry.MaxValue = ''; SubObjectsOfflineInfo.PDO Mapping Entry.AccessType = 'const';
            SubObjectsOfflineInfo.PDO Mapping Entry.IEC Variable = ''; SubObjectsOfflineInfo.PDO Mapping Entry.DefaultValue = '0x62000808'; SubObjectsOfflineInfo.PDO Mapping Entry.ObjectFlags = 16#00000000; SubObjectsOfflineInfo.Highest sub-index supported.Index = 16#00001800; SubObjectsOfflineInfo.Highest sub-index supported.SubIndex = 16#00; SubObjectsOfflineInfo.Highest sub-index supported.PDOMapping = FALSE; SubObjectsOfflineInfo.Highest sub-index supported.ObjectOwner = 16#03; SubObjectsOfflineInfo.Highest sub-index supported.ObjectType = 16#00000007; SubObjectsOfflineInfo.Highest sub-index supported.MinValue = '0x02'; SubObjectsOfflineInfo.Highest sub-index supported.MaxValue = '0x06'; SubObjectsOfflineInfo.Highest sub-index supported.AccessType = 'const'; SubObjectsOfflineInfo.Highest sub-index supported.IEC Variable = ''; SubObjectsOfflineInfo.Highest sub-index supported.DefaultValue = '0x5'; SubObjectsOfflineInfo.Highest sub-index supported.ObjectFlags = 16#00000000; SubObjectsOfflineInfo.COB-ID used by TPDO.Index = 16#00001800; SubObjectsOfflineInfo.COB-ID used by TPDO.SubIndex = 16#01; SubObjectsOfflineInfo.COB-ID used by TPDO.PDOMapping = FALSE; SubObjectsOfflineInfo.COB-ID used by TPDO.ObjectOwner = 16#03; SubObjectsOfflineInfo.COB-ID used by TPDO.ObjectType = 16#00000007; SubObjectsOfflineInfo.COB-ID used by TPDO.MinValue = '0x00000080'; SubObjectsOfflineInfo.COB-ID used by TPDO.MaxValue = '0xFFFFFFFF'; SubObjectsOfflineInfo.COB-ID used by TPDO.AccessType = 'rw'; SubObjectsOfflineInfo.COB-ID used by TPDO.IEC Variable = ''; SubObjectsOfflineInfo.COB-ID used by TPDO.DefaultValue = '$$NODEID+0x180'; SubObjectsOfflineInfo.COB-ID used by TPDO.ObjectFlags = 16#00000000; SubObjectsOfflineInfo.Transmission Type.Index = 16#00001800; SubObjectsOfflineInfo.Transmission Type.SubIndex = 16#02; SubObjectsOfflineInfo.Transmission Type.PDOMapping = FALSE; SubObjectsOfflineInfo.Transmission Type.ObjectOwner = 16#03; SubObjectsOfflineInfo.Transmission Type.ObjectType = 16#00000007; SubObjectsOfflineInfo.Transmission Type.MinValue = ''; SubObjectsOfflineInfo.Transmission Type.MaxValue = ''; SubObjectsOfflineInfo.Transmission Type.AccessType = 'rw'; SubObjectsOfflineInfo.Transmission Type.IEC Variable = ''; SubObjectsOfflineInfo.Transmission Type.DefaultValue = '0xFF'; SubObjectsOfflineInfo.Transmission Type.ObjectFlags = 16#00000000; SubObjectsOfflineInfo.Inhibit time.Index = 16#00001800; SubObjectsOfflineInfo.Inhibit time.SubIndex = 16#03; SubObjectsOfflineInfo.Inhibit time.PDOMapping = FALSE; SubObjectsOfflineInfo.Inhibit time.ObjectOwner = 16#03;
            SubObjectsOfflineInfo.Inhibit time.ObjectType = 16#00000007; SubObjectsOfflineInfo.Inhibit time.MinValue = ''; SubObjectsOfflineInfo.Inhibit time.MaxValue = ''; SubObjectsOfflineInfo.Inhibit time.AccessType = 'rw'; SubObjectsOfflineInfo.Inhibit time.IEC Variable = ''; SubObjectsOfflineInfo.Inhibit time.DefaultValue = '0x0'; SubObjectsOfflineInfo.Inhibit time.ObjectFlags = 16#00000000; SubObjectsOfflineInfo.compatibility entry.Index = 16#00001800; SubObjectsOfflineInfo.compatibility entry.SubIndex = 16#04; SubObjectsOfflineInfo.compatibility entry.PDOMapping = FALSE; SubObjectsOfflineInfo.compatibility entry.ObjectOwner = 16#03; SubObjectsOfflineInfo.compatibility entry.ObjectType = 16#00000007; SubObjectsOfflineInfo.compatibility entry.MinValue = ''; SubObjectsOfflineInfo.compatibility entry.MaxValue = ''; SubObjectsOfflineInfo.compatibility entry.AccessType = 'rw'; SubObjectsOfflineInfo.compatibility entry.IEC Variable = ''; SubObjectsOfflineInfo.compatibility entry.DefaultValue = '0x0'; SubObjectsOfflineInfo.compatibility entry.ObjectFlags = 16#00000000; SubObjectsOfflineInfo.Event timer.Index = 16#00001800; SubObjectsOfflineInfo.Event timer.SubIndex = 16#05; SubObjectsOfflineInfo.Event timer.PDOMapping = FALSE; SubObjectsOfflineInfo.Event timer.ObjectOwner = 16#03; SubObjectsOfflineInfo.Event timer.ObjectType = 16#00000007; SubObjectsOfflineInfo.Event timer.MinValue = ''; SubObjectsOfflineInfo.Event timer.MaxValue = ''; SubObjectsOfflineInfo.Event timer.AccessType = 'rw'; SubObjectsOfflineInfo.Event timer.IEC Variable = ''; SubObjectsOfflineInfo.Event timer.DefaultValue = '0x0'; SubObjectsOfflineInfo.Event timer.ObjectFlags = 16#00000000; SubObjectsOfflineInfo.Number of mapped application objects in TPDO.Index = 16#00001A00; SubObjectsOfflineInfo.Number of mapped application objects in TPDO.SubIndex = 16#00; SubObjectsOfflineInfo.Number of mapped application objects in TPDO.PDOMapping = FALSE; SubObjectsOfflineInfo.Number of mapped application objects in TPDO.ObjectOwner = 16#03; SubObjectsOfflineInfo.Number of mapped application objects in TPDO.ObjectType = 16#00000007; SubObjectsOfflineInfo.Number of mapped application objects in TPDO.MinValue = '0'; SubObjectsOfflineInfo.Number of mapped application objects in TPDO.MaxValue = '8'; SubObjectsOfflineInfo.Number of mapped application objects in TPDO.AccessType = 'const'; SubObjectsOfflineInfo.Number of mapped application objects in TPDO.IEC Variable = ''; SubObjectsOfflineInfo.Number of mapped application objects in TPDO.DefaultValue = '0x08'; SubObjectsOfflineInfo.Number of mapped application objects in TPDO.ObjectFlags = 16#00000000;
            SubObjectsOfflineInfo.PDO Mapping Entry.Index = 16#00001A00; SubObjectsOfflineInfo.PDO Mapping Entry.SubIndex = 16#01; SubObjectsOfflineInfo.PDO Mapping Entry.PDOMapping = FALSE; SubObjectsOfflineInfo.PDO Mapping Entry.ObjectOwner = 16#03; SubObjectsOfflineInfo.PDO Mapping Entry.ObjectType = 16#00000007; SubObjectsOfflineInfo.PDO Mapping Entry.MinValue = ''; SubObjectsOfflineInfo.PDO Mapping Entry.MaxValue = ''; SubObjectsOfflineInfo.PDO Mapping Entry.AccessType = 'const'; SubObjectsOfflineInfo.PDO Mapping Entry.IEC Variable = ''; SubObjectsOfflineInfo.PDO Mapping Entry.DefaultValue = '0x60000108'; SubObjectsOfflineInfo.PDO Mapping Entry.ObjectFlags = 16#00000000; SubObjectsOfflineInfo.PDO Mapping Entry.Index = 16#00001A00; SubObjectsOfflineInfo.PDO Mapping Entry.SubIndex = 16#02; SubObjectsOfflineInfo.PDO Mapping Entry.PDOMapping = FALSE; SubObjectsOfflineInfo.PDO Mapping Entry.ObjectOwner = 16#03; SubObjectsOfflineInfo.PDO Mapping Entry.ObjectType = 16#00000007; SubObjectsOfflineInfo.PDO Mapping Entry.MinValue = ''; SubObjectsOfflineInfo.PDO Mapping Entry.MaxValue = ''; SubObjectsOfflineInfo.PDO Mapping Entry.AccessType = 'const'; SubObjectsOfflineInfo.PDO Mapping Entry.IEC Variable = ''; SubObjectsOfflineInfo.PDO Mapping Entry.DefaultValue = '0x60000208'; SubObjectsOfflineInfo.PDO Mapping Entry.ObjectFlags = 16#00000000; SubObjectsOfflineInfo.PDO Mapping Entry.Index = 16#00001A00; SubObjectsOfflineInfo.PDO Mapping Entry.SubIndex = 16#03; SubObjectsOfflineInfo.PDO Mapping Entry.PDOMapping = FALSE; SubObjectsOfflineInfo.PDO Mapping Entry.ObjectOwner = 16#03; SubObjectsOfflineInfo.PDO Mapping Entry.ObjectType = 16#00000007; SubObjectsOfflineInfo.PDO Mapping Entry.MinValue = ''; SubObjectsOfflineInfo.PDO Mapping Entry.MaxValue = ''; SubObjectsOfflineInfo.PDO Mapping Entry.AccessType = 'const'; SubObjectsOfflineInfo.PDO Mapping Entry.IEC Variable = ''; SubObjectsOfflineInfo.PDO Mapping Entry.DefaultValue = '0x60000308'; SubObjectsOfflineInfo.PDO Mapping Entry.ObjectFlags = 16#00000000; SubObjectsOfflineInfo.PDO Mapping Entry.Index = 16#00001A00; SubObjectsOfflineInfo.PDO Mapping Entry.SubIndex = 16#04; SubObjectsOfflineInfo.PDO Mapping Entry.PDOMapping = FALSE; SubObjectsOfflineInfo.PDO Mapping Entry.ObjectOwner = 16#03; SubObjectsOfflineInfo.PDO Mapping Entry.ObjectType = 16#00000007; SubObjectsOfflineInfo.PDO Mapping Entry.MinValue = ''; SubObjectsOfflineInfo.PDO Mapping Entry.MaxValue = '';
            SubObjectsOfflineInfo.PDO Mapping Entry.AccessType = 'const'; SubObjectsOfflineInfo.PDO Mapping Entry.IEC Variable = ''; SubObjectsOfflineInfo.PDO Mapping Entry.DefaultValue = '0x60000408'; SubObjectsOfflineInfo.PDO Mapping Entry.ObjectFlags = 16#00000000; SubObjectsOfflineInfo.PDO Mapping Entry.Index = 16#00001A00; SubObjectsOfflineInfo.PDO Mapping Entry.SubIndex = 16#05; SubObjectsOfflineInfo.PDO Mapping Entry.PDOMapping = FALSE; SubObjectsOfflineInfo.PDO Mapping Entry.ObjectOwner = 16#03; SubObjectsOfflineInfo.PDO Mapping Entry.ObjectType = 16#00000007; SubObjectsOfflineInfo.PDO Mapping Entry.MinValue = ''; SubObjectsOfflineInfo.PDO Mapping Entry.MaxValue = ''; SubObjectsOfflineInfo.PDO Mapping Entry.AccessType = 'const'; SubObjectsOfflineInfo.PDO Mapping Entry.IEC Variable = ''; SubObjectsOfflineInfo.PDO Mapping Entry.DefaultValue = '0x60000508'; SubObjectsOfflineInfo.PDO Mapping Entry.ObjectFlags = 16#00000000; SubObjectsOfflineInfo.PDO Mapping Entry.Index = 16#00001A00; SubObjectsOfflineInfo.PDO Mapping Entry.SubIndex = 16#06; SubObjectsOfflineInfo.PDO Mapping Entry.PDOMapping = FALSE; SubObjectsOfflineInfo.PDO Mapping Entry.ObjectOwner = 16#03; SubObjectsOfflineInfo.PDO Mapping Entry.ObjectType = 16#00000007; SubObjectsOfflineInfo.PDO Mapping Entry.MinValue = ''; SubObjectsOfflineInfo.PDO Mapping Entry.MaxValue = ''; SubObjectsOfflineInfo.PDO Mapping Entry.AccessType = 'const'; SubObjectsOfflineInfo.PDO Mapping Entry.IEC Variable = ''; SubObjectsOfflineInfo.PDO Mapping Entry.DefaultValue = '0x60000608'; SubObjectsOfflineInfo.PDO Mapping Entry.ObjectFlags = 16#00000000; SubObjectsOfflineInfo.PDO Mapping Entry.Index = 16#00001A00; SubObjectsOfflineInfo.PDO Mapping Entry.SubIndex = 16#07; SubObjectsOfflineInfo.PDO Mapping Entry.PDOMapping = FALSE; SubObjectsOfflineInfo.PDO Mapping Entry.ObjectOwner = 16#03; SubObjectsOfflineInfo.PDO Mapping Entry.ObjectType = 16#00000007; SubObjectsOfflineInfo.PDO Mapping Entry.MinValue = ''; SubObjectsOfflineInfo.PDO Mapping Entry.MaxValue = ''; SubObjectsOfflineInfo.PDO Mapping Entry.AccessType = 'const'; SubObjectsOfflineInfo.PDO Mapping Entry.IEC Variable = ''; SubObjectsOfflineInfo.PDO Mapping Entry.DefaultValue = '0x60000708'; SubObjectsOfflineInfo.PDO Mapping Entry.ObjectFlags = 16#00000000; SubObjectsOfflineInfo.PDO Mapping Entry.Index = 16#00001A00; SubObjectsOfflineInfo.PDO Mapping Entry.SubIndex = 16#08; SubObjectsOfflineInfo.PDO Mapping Entry.PDOMapping = FALSE;
            SubObjectsOfflineInfo.PDO Mapping Entry.ObjectOwner = 16#03; SubObjectsOfflineInfo.PDO Mapping Entry.ObjectType = 16#00000007; SubObjectsOfflineInfo.PDO Mapping Entry.MinValue = ''; SubObjectsOfflineInfo.PDO Mapping Entry.MaxValue = ''; SubObjectsOfflineInfo.PDO Mapping Entry.AccessType = 'const'; SubObjectsOfflineInfo.PDO Mapping Entry.IEC Variable = ''; SubObjectsOfflineInfo.PDO Mapping Entry.DefaultValue = '0x60000808'; SubObjectsOfflineInfo.PDO Mapping Entry.ObjectFlags = 16#00000000; SubObjectsOfflineInfo.TestString.Index = 16#00003000; SubObjectsOfflineInfo.TestString.SubIndex = 16#00; SubObjectsOfflineInfo.TestString.PDOMapping = FALSE; SubObjectsOfflineInfo.TestString.ObjectOwner = 16#03; SubObjectsOfflineInfo.TestString.ObjectType = 16#00000007; SubObjectsOfflineInfo.TestString.MinValue = ''; SubObjectsOfflineInfo.TestString.MaxValue = ''; SubObjectsOfflineInfo.TestString.AccessType = 'rw'; SubObjectsOfflineInfo.TestString.IEC Variable = 'CANopenLocalDeviceExamples.strTestString'; SubObjectsOfflineInfo.TestString.DefaultValue = ''; SubObjectsOfflineInfo.TestString.ObjectFlags = 16#00000000; SubObjectsOfflineInfo.Number of Elements.Index = 16#00006000; SubObjectsOfflineInfo.Number of Elements.SubIndex = 16#00; SubObjectsOfflineInfo.Number of Elements.PDOMapping = FALSE; SubObjectsOfflineInfo.Number of Elements.ObjectOwner = 16#03; SubObjectsOfflineInfo.Number of Elements.ObjectType = 16#00000007; SubObjectsOfflineInfo.Number of Elements.MinValue = ''; SubObjectsOfflineInfo.Number of Elements.MaxValue = ''; SubObjectsOfflineInfo.Number of Elements.AccessType = 'ro'; SubObjectsOfflineInfo.Number of Elements.IEC Variable = ''; SubObjectsOfflineInfo.Number of Elements.DefaultValue = '0x8'; SubObjectsOfflineInfo.Number of Elements.ObjectFlags = 16#00000000; SubObjectsOfflineInfo.DigInput8.Index = 16#00006000; SubObjectsOfflineInfo.DigInput8.SubIndex = 16#01; SubObjectsOfflineInfo.DigInput8.PDOMapping = TRUE; SubObjectsOfflineInfo.DigInput8.ObjectOwner = 16#03; SubObjectsOfflineInfo.DigInput8.ObjectType = 16#00000007; SubObjectsOfflineInfo.DigInput8.MinValue = ''; SubObjectsOfflineInfo.DigInput8.MaxValue = ''; SubObjectsOfflineInfo.DigInput8.AccessType = 'ro'; SubObjectsOfflineInfo.DigInput8.IEC Variable = ''; SubObjectsOfflineInfo.DigInput8.DefaultValue = '';
            SubObjectsOfflineInfo.DigInput8.ObjectFlags = 16#00000000; SubObjectsOfflineInfo.DigInput8.Index = 16#00006000; SubObjectsOfflineInfo.DigInput8.SubIndex = 16#02; SubObjectsOfflineInfo.DigInput8.PDOMapping = TRUE; SubObjectsOfflineInfo.DigInput8.ObjectOwner = 16#03; SubObjectsOfflineInfo.DigInput8.ObjectType = 16#00000007; SubObjectsOfflineInfo.DigInput8.MinValue = ''; SubObjectsOfflineInfo.DigInput8.MaxValue = ''; SubObjectsOfflineInfo.DigInput8.AccessType = 'ro'; SubObjectsOfflineInfo.DigInput8.IEC Variable = ''; SubObjectsOfflineInfo.DigInput8.DefaultValue = ''; SubObjectsOfflineInfo.DigInput8.ObjectFlags = 16#00000000; SubObjectsOfflineInfo.DigInput8.Index = 16#00006000; SubObjectsOfflineInfo.DigInput8.SubIndex = 16#03; SubObjectsOfflineInfo.DigInput8.PDOMapping = TRUE; SubObjectsOfflineInfo.DigInput8.ObjectOwner = 16#03; SubObjectsOfflineInfo.DigInput8.ObjectType = 16#00000007; SubObjectsOfflineInfo.DigInput8.MinValue = ''; SubObjectsOfflineInfo.DigInput8.MaxValue = ''; SubObjectsOfflineInfo.DigInput8.AccessType = 'ro'; SubObjectsOfflineInfo.DigInput8.IEC Variable = ''; SubObjectsOfflineInfo.DigInput8.DefaultValue = ''; SubObjectsOfflineInfo.DigInput8.ObjectFlags = 16#00000000; SubObjectsOfflineInfo.DigInput8.Index = 16#00006000; SubObjectsOfflineInfo.DigInput8.SubIndex = 16#04; SubObjectsOfflineInfo.DigInput8.PDOMapping = TRUE; SubObjectsOfflineInfo.DigInput8.ObjectOwner = 16#03; SubObjectsOfflineInfo.DigInput8.ObjectType = 16#00000007; SubObjectsOfflineInfo.DigInput8.MinValue = ''; SubObjectsOfflineInfo.DigInput8.MaxValue = ''; SubObjectsOfflineInfo.DigInput8.AccessType = 'ro'; SubObjectsOfflineInfo.DigInput8.IEC Variable = ''; SubObjectsOfflineInfo.DigInput8.DefaultValue = ''; SubObjectsOfflineInfo.DigInput8.ObjectFlags = 16#00000000; SubObjectsOfflineInfo.DigInput8.Index = 16#00006000; SubObjectsOfflineInfo.DigInput8.SubIndex = 16#05; SubObjectsOfflineInfo.DigInput8.PDOMapping = TRUE; SubObjectsOfflineInfo.DigInput8.ObjectOwner = 16#03; SubObjectsOfflineInfo.DigInput8.ObjectType = 16#00000007; SubObjectsOfflineInfo.DigInput8.MinValue = '';
            SubObjectsOfflineInfo.DigInput8.MaxValue = ''; SubObjectsOfflineInfo.DigInput8.AccessType = 'ro'; SubObjectsOfflineInfo.DigInput8.IEC Variable = ''; SubObjectsOfflineInfo.DigInput8.DefaultValue = ''; SubObjectsOfflineInfo.DigInput8.ObjectFlags = 16#00000000; SubObjectsOfflineInfo.DigInput8.Index = 16#00006000; SubObjectsOfflineInfo.DigInput8.SubIndex = 16#06; SubObjectsOfflineInfo.DigInput8.PDOMapping = TRUE; SubObjectsOfflineInfo.DigInput8.ObjectOwner = 16#03; SubObjectsOfflineInfo.DigInput8.ObjectType = 16#00000007; SubObjectsOfflineInfo.DigInput8.MinValue = ''; SubObjectsOfflineInfo.DigInput8.MaxValue = ''; SubObjectsOfflineInfo.DigInput8.AccessType = 'ro'; SubObjectsOfflineInfo.DigInput8.IEC Variable = ''; SubObjectsOfflineInfo.DigInput8.DefaultValue = ''; SubObjectsOfflineInfo.DigInput8.ObjectFlags = 16#00000000; SubObjectsOfflineInfo.DigInput8.Index = 16#00006000; SubObjectsOfflineInfo.DigInput8.SubIndex = 16#07; SubObjectsOfflineInfo.DigInput8.PDOMapping = TRUE; SubObjectsOfflineInfo.DigInput8.ObjectOwner = 16#03; SubObjectsOfflineInfo.DigInput8.ObjectType = 16#00000007; SubObjectsOfflineInfo.DigInput8.MinValue = ''; SubObjectsOfflineInfo.DigInput8.MaxValue = ''; SubObjectsOfflineInfo.DigInput8.AccessType = 'ro'; SubObjectsOfflineInfo.DigInput8.IEC Variable = ''; SubObjectsOfflineInfo.DigInput8.DefaultValue = ''; SubObjectsOfflineInfo.DigInput8.ObjectFlags = 16#00000000; SubObjectsOfflineInfo.DigInput8.Index = 16#00006000; SubObjectsOfflineInfo.DigInput8.SubIndex = 16#08; SubObjectsOfflineInfo.DigInput8.PDOMapping = TRUE; SubObjectsOfflineInfo.DigInput8.ObjectOwner = 16#03; SubObjectsOfflineInfo.DigInput8.ObjectType = 16#00000007; SubObjectsOfflineInfo.DigInput8.MinValue = ''; SubObjectsOfflineInfo.DigInput8.MaxValue = ''; SubObjectsOfflineInfo.DigInput8.AccessType = 'ro'; SubObjectsOfflineInfo.DigInput8.IEC Variable = ''; SubObjectsOfflineInfo.DigInput8.DefaultValue = ''; SubObjectsOfflineInfo.DigInput8.ObjectFlags = 16#00000000; SubObjectsOfflineInfo.Number of Elements.Index = 16#00006200; SubObjectsOfflineInfo.Number of Elements.SubIndex = 16#00;
            SubObjectsOfflineInfo.Number of Elements.PDOMapping = FALSE; SubObjectsOfflineInfo.Number of Elements.ObjectOwner = 16#03; SubObjectsOfflineInfo.Number of Elements.ObjectType = 16#00000007; SubObjectsOfflineInfo.Number of Elements.MinValue = ''; SubObjectsOfflineInfo.Number of Elements.MaxValue = ''; SubObjectsOfflineInfo.Number of Elements.AccessType = 'ro'; SubObjectsOfflineInfo.Number of Elements.IEC Variable = ''; SubObjectsOfflineInfo.Number of Elements.DefaultValue = '0x8'; SubObjectsOfflineInfo.Number of Elements.ObjectFlags = 16#00000000; SubObjectsOfflineInfo.DigOutput8.Index = 16#00006200; SubObjectsOfflineInfo.DigOutput8.SubIndex = 16#01; SubObjectsOfflineInfo.DigOutput8.PDOMapping = TRUE; SubObjectsOfflineInfo.DigOutput8.ObjectOwner = 16#03; SubObjectsOfflineInfo.DigOutput8.ObjectType = 16#00000007; SubObjectsOfflineInfo.DigOutput8.MinValue = ''; SubObjectsOfflineInfo.DigOutput8.MaxValue = ''; SubObjectsOfflineInfo.DigOutput8.AccessType = 'rww'; SubObjectsOfflineInfo.DigOutput8.IEC Variable = ''; SubObjectsOfflineInfo.DigOutput8.DefaultValue = '0'; SubObjectsOfflineInfo.DigOutput8.ObjectFlags = 16#00000000; SubObjectsOfflineInfo.DigOutput8.Index = 16#00006200; SubObjectsOfflineInfo.DigOutput8.SubIndex = 16#02; SubObjectsOfflineInfo.DigOutput8.PDOMapping = TRUE; SubObjectsOfflineInfo.DigOutput8.ObjectOwner = 16#03; SubObjectsOfflineInfo.DigOutput8.ObjectType = 16#00000007; SubObjectsOfflineInfo.DigOutput8.MinValue = ''; SubObjectsOfflineInfo.DigOutput8.MaxValue = ''; SubObjectsOfflineInfo.DigOutput8.AccessType = 'rww'; SubObjectsOfflineInfo.DigOutput8.IEC Variable = ''; SubObjectsOfflineInfo.DigOutput8.DefaultValue = '0'; SubObjectsOfflineInfo.DigOutput8.ObjectFlags = 16#00000000; SubObjectsOfflineInfo.DigOutput8.Index = 16#00006200; SubObjectsOfflineInfo.DigOutput8.SubIndex = 16#03; SubObjectsOfflineInfo.DigOutput8.PDOMapping = TRUE; SubObjectsOfflineInfo.DigOutput8.ObjectOwner = 16#03; SubObjectsOfflineInfo.DigOutput8.ObjectType = 16#00000007; SubObjectsOfflineInfo.DigOutput8.MinValue = ''; SubObjectsOfflineInfo.DigOutput8.MaxValue = ''; SubObjectsOfflineInfo.DigOutput8.AccessType = 'rww'; SubObjectsOfflineInfo.DigOutput8.IEC Variable = '';
            SubObjectsOfflineInfo.DigOutput8.DefaultValue = '0'; SubObjectsOfflineInfo.DigOutput8.ObjectFlags = 16#00000000; SubObjectsOfflineInfo.DigOutput8.Index = 16#00006200; SubObjectsOfflineInfo.DigOutput8.SubIndex = 16#04; SubObjectsOfflineInfo.DigOutput8.PDOMapping = TRUE; SubObjectsOfflineInfo.DigOutput8.ObjectOwner = 16#03; SubObjectsOfflineInfo.DigOutput8.ObjectType = 16#00000007; SubObjectsOfflineInfo.DigOutput8.MinValue = ''; SubObjectsOfflineInfo.DigOutput8.MaxValue = ''; SubObjectsOfflineInfo.DigOutput8.AccessType = 'rww'; SubObjectsOfflineInfo.DigOutput8.IEC Variable = ''; SubObjectsOfflineInfo.DigOutput8.DefaultValue = '0'; SubObjectsOfflineInfo.DigOutput8.ObjectFlags = 16#00000000; SubObjectsOfflineInfo.DigOutput8.Index = 16#00006200; SubObjectsOfflineInfo.DigOutput8.SubIndex = 16#05; SubObjectsOfflineInfo.DigOutput8.PDOMapping = TRUE; SubObjectsOfflineInfo.DigOutput8.ObjectOwner = 16#03; SubObjectsOfflineInfo.DigOutput8.ObjectType = 16#00000007; SubObjectsOfflineInfo.DigOutput8.MinValue = ''; SubObjectsOfflineInfo.DigOutput8.MaxValue = ''; SubObjectsOfflineInfo.DigOutput8.AccessType = 'rww'; SubObjectsOfflineInfo.DigOutput8.IEC Variable = ''; SubObjectsOfflineInfo.DigOutput8.DefaultValue = '0'; SubObjectsOfflineInfo.DigOutput8.ObjectFlags = 16#00000000; SubObjectsOfflineInfo.DigOutput8.Index = 16#00006200; SubObjectsOfflineInfo.DigOutput8.SubIndex = 16#06; SubObjectsOfflineInfo.DigOutput8.PDOMapping = TRUE; SubObjectsOfflineInfo.DigOutput8.ObjectOwner = 16#03; SubObjectsOfflineInfo.DigOutput8.ObjectType = 16#00000007; SubObjectsOfflineInfo.DigOutput8.MinValue = ''; SubObjectsOfflineInfo.DigOutput8.MaxValue = ''; SubObjectsOfflineInfo.DigOutput8.AccessType = 'rww'; SubObjectsOfflineInfo.DigOutput8.IEC Variable = ''; SubObjectsOfflineInfo.DigOutput8.DefaultValue = '0'; SubObjectsOfflineInfo.DigOutput8.ObjectFlags = 16#00000000; SubObjectsOfflineInfo.DigOutput8.Index = 16#00006200; SubObjectsOfflineInfo.DigOutput8.SubIndex = 16#07; SubObjectsOfflineInfo.DigOutput8.PDOMapping = TRUE; SubObjectsOfflineInfo.DigOutput8.ObjectOwner = 16#03; SubObjectsOfflineInfo.DigOutput8.ObjectType = 16#00000007;
            SubObjectsOfflineInfo.DigOutput8.MinValue = ''; SubObjectsOfflineInfo.DigOutput8.MaxValue = ''; SubObjectsOfflineInfo.DigOutput8.AccessType = 'rww'; SubObjectsOfflineInfo.DigOutput8.IEC Variable = ''; SubObjectsOfflineInfo.DigOutput8.DefaultValue = '0'; SubObjectsOfflineInfo.DigOutput8.ObjectFlags = 16#00000000; SubObjectsOfflineInfo.DigOutput8.Index = 16#00006200; SubObjectsOfflineInfo.DigOutput8.SubIndex = 16#08; SubObjectsOfflineInfo.DigOutput8.PDOMapping = TRUE; SubObjectsOfflineInfo.DigOutput8.ObjectOwner = 16#03; SubObjectsOfflineInfo.DigOutput8.ObjectType = 16#00000007; SubObjectsOfflineInfo.DigOutput8.MinValue = ''; SubObjectsOfflineInfo.DigOutput8.MaxValue = ''; SubObjectsOfflineInfo.DigOutput8.AccessType = 'rww'; SubObjectsOfflineInfo.DigOutput8.IEC Variable = ''; SubObjectsOfflineInfo.DigOutput8.DefaultValue = '0'; SubObjectsOfflineInfo.DigOutput8.ObjectFlags = 16#00000000; SubObjectsOfflineInfo.Number of Elements.Index = 16#00006412; SubObjectsOfflineInfo.Number of Elements.SubIndex = 16#00; SubObjectsOfflineInfo.Number of Elements.PDOMapping = FALSE; SubObjectsOfflineInfo.Number of Elements.ObjectOwner = 16#03; SubObjectsOfflineInfo.Number of Elements.ObjectType = 16#00000007; SubObjectsOfflineInfo.Number of Elements.MinValue = ''; SubObjectsOfflineInfo.Number of Elements.MaxValue = ''; SubObjectsOfflineInfo.Number of Elements.AccessType = 'ro'; SubObjectsOfflineInfo.Number of Elements.IEC Variable = ''; SubObjectsOfflineInfo.Number of Elements.DefaultValue = '0x1'; SubObjectsOfflineInfo.Number of Elements.ObjectFlags = 16#00000000; SubObjectsOfflineInfo.AnalogueOutput32.Index = 16#00006412; SubObjectsOfflineInfo.AnalogueOutput32.SubIndex = 16#01; SubObjectsOfflineInfo.AnalogueOutput32.PDOMapping = FALSE; SubObjectsOfflineInfo.AnalogueOutput32.ObjectOwner = 16#03; SubObjectsOfflineInfo.AnalogueOutput32.ObjectType = 16#00000007; SubObjectsOfflineInfo.AnalogueOutput32.MinValue = ''; SubObjectsOfflineInfo.AnalogueOutput32.MaxValue = ''; SubObjectsOfflineInfo.AnalogueOutput32.AccessType = 'rww'; SubObjectsOfflineInfo.AnalogueOutput32.IEC Variable = ''; SubObjectsOfflineInfo.AnalogueOutput32.DefaultValue = '0'; SubObjectsOfflineInfo.AnalogueOutput32.ObjectFlags = 16#00000000; 1008sub00_Data = ['CANopenDeviceExample'];
            3000sub00_Data = ['']
          unmapped channels: DigInput8, DigInput8, DigInput8, DigInput8, DigInput8, DigInput8, DigInput8, DigInput8, DigOutput8, DigOutput8, DigOutput8, DigOutput8, DigOutput8, DigOutput8, DigOutput8, DigOutput8
  00000000-0000-0000-0000-000000000000|C:\Users\m.lamp\Documents\license.txt
*)

// Device/Application/CANopen Slave Examples/Network management/NMT_Command
{attribute 'qualified_only'}
{attribute 'strict'}
TYPE NMT_Command :
(
	RESET,
	START,
	STOP,
	PREOP,
	POWER_DOWN,
	POWER_UP
);
END_TYPE

// Device/Application/CANopen Master Examples/CANopenManagerExamples
PROGRAM CANopenManagerExamples
VAR
END_VAR

///////////////////////////////////////// CIA 405 Examples //////////////////////////////////////////////////////

//Diagnosis Examples
GetStateExample(); //How to get the state of a CANopenRemote Device?
GetCANopenKernelStateExample(); //How to get the CANopen stack kernel state?
ReceiveEMCYFromAllDevicesExample(); //How to check if any CANopenRemote Device has a pending Emergency?
ReceiveEMCYFromOneDeviceExample(); //How to check if a specific CANopenRemote Device has a pending Emergency?

//SDO Examples
ExpeditedReadExample(); //How to read up to 4 bytes by SDO?
ExpeditedWriteExample(); //How to write up to 4 bytes by SDO?
SegmentedAndBlockReadExample(); //How to read more than 4 bytes by SDO?
SegmentedAndBlockWriteExample(); //How to write more than 4 bytes by SDO?

NMT_Example(); //How to start/stop/reset CANopenRemote Devices?

GetCANopenManagerNodeIDExample(); //How to read the CANopen Manager NodeID?

///////////////////////////////////////// General Examples //////////////////////////////////////////////////////

CANopenManagerAPI(); //How to use the CANopen Manager API?
CANopenRemoteDeviceAPI(); //How to use the CANopenRemoteDevice API?

END_PROGRAM

// Device/Application/CANopen Master Examples/CiA405/Diagnosis/State/GetStateExample
// The following program gets the current CANopen state of the CANopenRemoteDevice attached below the CANopen_Manager.
// Set xEnable to TRUE in online mode to get the program working.
PROGRAM GetStateExample
VAR
	xEnable : BOOL; // Set this variable to true to start the example code. Variable will be set to FALSE if GetState finished execution.
	State : CiA405.DEVICE_STATE; // Result: CANopen State
	
	GetState : CIA405.GET_STATE;
END_VAR

IF GetState.CONFIRM = TRUE THEN
	// GetState successful. Output STATE contains result.
	State := GetState.STATE;
	xEnable := FALSE;
ELSIF GetState.ERROR <> CIA405.CANOPEN_KERNEL_ERROR.CANOPEN_KERNEL_NO_ERROR THEN
	// an error occured while processing GetState e.g. wrong NodeID or NetworkID
	xEnable := FALSE;
END_IF

// GetState needs the CAN network and the device NodeID (input DEVICE). 
GetState( 	ENABLE := xEnable,
		  	NETWORK := CANbus.NetId + 1, //CODESYS NetId starts by 0 (the number entered into the CANbus configurator); CiA405 NETWORK by 1; That is the reason why we have to increment it here.
		  	TIMEOUT := 0, // no timeout for GetState needed because it is processed locally.
			DEVICE := CANopenRemoteDevice.NodeID // Note: If you want to get the state of the CANopenManager, you can use the CANopenManager NodeID or NodeID 0.
												 // A CANopenManager goes to OPERATIONAL if all mandatory (= not optional) slaves are operational.
);

END_PROGRAM

// Device/Application/CANopen Master Examples/CiA405/Diagnosis/State/GetCANopenKernelStateExample
// This program gets the state of the CANopenManager kernel. If kernel has no error everything is working fine.
// See CiA405.CANOPEN_KERNEL_ERROR in library manager for further details.
// Set xEnable to TRUE in online mode to get the program working.
PROGRAM GetCANopenKernelStateExample
VAR
	xEnable : BOOL; // Set this variable to true to start the example code. Variable will be set to FALSE if GetState finished execution.
	xErrorPending : BOOL; //true if a CANopen Kernel error is pending
	State : CiA405.CANOPEN_KERNEL_ERROR; // Result: CANopen Manager kernel state
	
	GetKernelState : CIA405.GET_CANOPEN_KERNEL_STATE;
END_VAR

IF GetKernelState.CONFIRM = TRUE THEN
	// GetKernelState successful. Output STATE contains result.
	State := GetKernelState.STATE;
	xErrorPending := State <> CIA405.CANOPEN_KERNEL_ERROR.CANOPEN_KERNEL_NO_ERROR;
	xEnable := FALSE;
ELSIF GetKernelState.ERROR <> CIA405.CANOPEN_KERNEL_ERROR.CANOPEN_KERNEL_NO_ERROR THEN
	// an error occured while processing GetKernelState e.g. wrong NetworkID
	xEnable := FALSE;
END_IF

GetKernelState( 	ENABLE := xEnable,
		  			NETWORK := CANbus.NetId + 1, //CODESYS NetId starts by 0 (the number entered into the CANbus configurator); CiA405 NETWORK by 1; That is the reason why we have to increment it here.
		  			TIMEOUT := 0 // no timeout for GetKernelState needed because it is processed locally.
);

END_PROGRAM

// Device/Application/CANopen Master Examples/CiA405/Diagnosis/EMCY/ReceiveEMCYFromAllDevicesExample
// This program checks if any emergency is pending for any device of a given CANopenManager network.
// Set xEnable to TRUE in online mode to get the program working.
PROGRAM ReceiveEMCYFromAllDevicesExample
VAR
	xEnable : BOOL; // Set this variable to true to start the example code. Variable will be set to FALSE if RecvEMCY finished execution.
	xEMCYPending : BOOL; //true if EMCY is pending ==> see EMCY and NodeID for EMCY information
	EMCY : CIA405.EMCY_ERROR; //contains EMCY information
	NodeID : CIA405.DEVICE; //NodeID of EMCY sender
	
	RecvEMCY : CIA405.RECV_EMCY;
END_VAR

IF RecvEMCY.CONFIRM = TRUE THEN
	// RecvEMCY successful.
	IF RecvEMCY.DEVICE <> 0 THEN
		//an EMCY from NodeID RecvEMCY.DEVICE is pending
		xEMCYPending := TRUE;
		EMCY := RecvEMCY.ERRORINFO;
		NodeID := RecvEMCY.DEVICE;
	ELSE
		//all devices are error free
		xEMCYPending := FALSE;
	END_IF

	xEnable := FALSE;
ELSIF RecvEMCY.ERROR <> CIA405.CANOPEN_KERNEL_ERROR.CANOPEN_KERNEL_NO_ERROR THEN
	// an error occured while processing RecvEMCY e.g. wrong NodeID or NetworkID
	xEnable := FALSE;
END_IF

RecvEMCY( 	ENABLE := xEnable,
		  	NETWORK := CANbus.NetId + 1, //CODESYS NetId starts by 0 (the number entered into the CANbus configurator); CiA405 NETWORK by 1; That is the reason why we have to increment it here.
		  	TIMEOUT := 0 // no timeout for RecvEMCY needed because it is processed locally.
);

END_PROGRAM

// Device/Application/CANopen Master Examples/CiA405/Diagnosis/EMCY/ReceiveEMCYFromOneDeviceExample
// This program checks if any emergency is pending for CANopenRemoteDevice.
// Set xEnable to TRUE in online mode to get the program working.
PROGRAM ReceiveEMCYFromOneDeviceExample
VAR
	xEnable : BOOL; // Set this variable to true to start the example code. Variable will be set to FALSE if RecvEMCYDev finished execution.
	xEMCYPending : BOOL; //true if EMCY is pending ==> see EMCY for EMCY information
	EMCY : CIA405.EMCY_ERROR; //contains EMCY information
	
	RecvEMCYDev : CIA405.RECV_EMCY_DEV;
END_VAR

IF RecvEMCYDev.CONFIRM = TRUE THEN
	// RecvEMCYDev successful
	IF RecvEMCYDev.ERRORINFO.EMCY_ERROR_CODE <> 0 THEN
		//an EMCY is pending ==> see RecvEMCYDev.ERRORINFO for EMCY information
		xEMCYPending := TRUE;
		EMCY := RecvEMCYDev.ERRORINFO;
	ELSE
		//device is error free
		xEMCYPending := FALSE;
	END_IF
	xEnable := FALSE;
ELSIF RecvEMCYDev.ERROR <> CIA405.CANOPEN_KERNEL_ERROR.CANOPEN_KERNEL_NO_ERROR THEN
	// an error occured while processing RecvEMCY e.g. wrong NodeID or NetworkID
	xEnable := FALSE;
END_IF

RecvEMCYDev( 	ENABLE := xEnable,
		  		NETWORK := CANbus.NetId + 1, //CODESYS NetId starts by 0 (the number entered into the CANbus configurator); CiA405 NETWORK by 1; That is the reason why we have to increment it here.
		  		TIMEOUT := 0, // no timeout for RecvEMCYDev needed because it is processed locally.
				DEVICE := CANopenRemoteDevice.NodeID //NodeID to receive EMCY from
);

END_PROGRAM

// Device/Application/CANopen Master Examples/CiA405/SDO access/Expedited (<= 4byte)/ExpeditedReadExample
// The following program reads the device type of CANopenRemoteDevice and shows how to usde SDORead4 function block.
// Set xEnable to TRUE in online mode to get the program working.
PROGRAM ExpeditedReadExample
VAR
	xEnable       : BOOL; // Set this variable to true to start the example code. Variable will be set to FALSE if Expedited transfer finished execution.
	dwValue : DWORD; //read value
	dwAbortCode : DWORD; //contains abort code in case of error
	
	SDORead4 	  : CIA405.SDO_READ4;
END_VAR

IF SDORead4.CONFIRM THEN
	//value was read without error
	// ==> Copy data from SDO read function block
	MEMUtils.MemCpy(pbyDest := ADR(dwValue), pbySrc := ADR(SDORead4.DATA[1]), dwSize := SIZEOF(dwValue));
	//==> On big endian systems: dwValue has to be swapped to CANopen byte order (= Little Endian).
	MEMUtils.SwapLocalToIntel(pAddress := ADR(dwValue), iSize := TO_INT(SIZEOF(dwValue))); //function only swaps on big endian systems
	xEnable := FALSE;
ELSIF SDORead4.ERROR <> CiA405.CANOPEN_KERNEL_ERROR.CANOPEN_KERNEL_NO_ERROR THEN
	//Error occured
	IF SDORead4.ERROR = CIA405.CANOPEN_KERNEL_ERROR.CANOPEN_KERNEL_OTHER_ERROR THEN
		//output error info contains abort code in little endian format
		MEMUtils.MemCpy(pbyDest := ADR(dwAbortCode), pbySrc := ADR(SDORead4.ERRORINFO), dwSize := SIZEOF(dwAbortCode));
		MEMUtils.SwapLocalToIntel(pAddress := ADR(dwAbortCode), iSize := TO_INT(SIZEOF(dwAbortCode))); //function only swaps on big endian systems	
	END_IF
	xEnable := FALSE;
END_IF

SDORead4(
	NETWORK:= CANbus.NetId + 1, //CODESYS NetId starts by 0 (the number entered into the CANbus configurator); CiA405 NETWORK by 1; That is the reason why we have to increment it here.
	ENABLE:= xEnable,
	TIMEOUT:= 0, //Timeout for SDO read in ms. Here: 0 ==> no timeout
	DEVICE:= CANopenRemoteDevice.NodeID, // NodeID of destination device
	CHANNEL:= 0, //SDO channel which should be used. 0 means auto channeling ==> the next free channel will be used. It depends on the slave which settings are working here but 0 and channel 1 is always working. 
	INDEX:= 16#1000, //object index which should be read
	SUBINDEX:= 0 //object sub index which should be read
);

END_PROGRAM

// Device/Application/CANopen Master Examples/CiA405/SDO access/Expedited (<= 4byte)/ExpeditedWriteExample
// The following program writes a 32bit value with SDO expedited transfer.
// Set xEnable to TRUE in online mode to get the program working.
PROGRAM ExpeditedWriteExample
VAR
	xEnable       : BOOL; // Set this variable to true to start the example code. Variable will be set to FALSE if Expedited transfer finished execution.
	diValue : DINT := 10; //value which should be written
	dwAbortCode : DWORD; //contains abort code in case of error
	
	SDOWrite4 	  : CiA405.SDO_WRITE4;
	RTrig 		  : Standard.R_TRIG;
END_VAR

RTrig(CLK := xEnable); //detect a rising edge for xEnable

IF RTrig.Q THEN
	// Rising edge for xEnable detected ==> Prepare SDO write function block
	// ==> Copy data to SDO write function block
	MEMUtils.MemCpy(pbyDest := ADR(SDOWrite4.DATA[1]), pbySrc := ADR(diValue), dwSize := SIZEOF(diValue));
	//==> On big endian systems: diValue has to be swapped to CANopen byte order (= Little Endian).
	MEMUtils.SwapLocalToIntel(pAddress := ADR(SDOWrite4.DATA[1]), iSize := TO_INT(SIZEOF(diValue))); //function only swaps on big endian systems
END_IF

IF SDOWrite4.CONFIRM THEN
	//value was written without error
	xEnable := FALSE;
ELSIF SDOWrite4.ERROR <> CiA405.CANOPEN_KERNEL_ERROR.CANOPEN_KERNEL_NO_ERROR THEN
	//Error occured
	IF SDOWrite4.ERROR = CIA405.CANOPEN_KERNEL_ERROR.CANOPEN_KERNEL_OTHER_ERROR THEN
		//output error info contains abort code in little endian format
		MEMUtils.MemCpy(pbyDest := ADR(dwAbortCode), pbySrc := ADR(SDOWrite4.ERRORINFO), dwSize := SIZEOF(dwAbortCode));
		MEMUtils.SwapLocalToIntel(pAddress := ADR(dwAbortCode), iSize := TO_INT(SIZEOF(dwAbortCode))); //function only swaps on big endian systems	
	END_IF
	xEnable := FALSE;
END_IF

SDOWrite4(
	NETWORK:= CANbus.NetId + 1, //CODESYS NetId starts by 0 (the number entered into the CANbus configurator); CiA405 NETWORK by 1; That is the reason why we have to increment it here.
	ENABLE:= xEnable,
	TIMEOUT:= 0, //Timeout for SDO write in ms. Here: 0 ==> no timeout
	DEVICE:= CANopenRemoteDevice.NodeID, // NodeID of destination device
	CHANNEL:= 0, //SDO channel which should be used. 0 means auto channeling ==> the next free channel will be used. It depends on the slave which settings are working here but 0 and channel 1 is always working. 
	INDEX:= 16#6412, //object index which should be written
	SUBINDEX:= 1, //object sub index which should be written
	DATALENGTH:= TO_USINT(SIZEOF(diValue)) //length of data to be written
);

END_PROGRAM

// Device/Application/CANopen Master Examples/CiA405/SDO access/Block and Segmented/SegmentedAndBlockReadExample
// This program uses CiA405.SDO_READ_DATA for reading more than 4 byte from a slave using segmented or block transfer.
//
// This example code reads object 16#1008sub0 which is the device name.
// CiA405.SDO_READ_DATA is a universal function block which can be also used for expedited transfer (<= 4byte).
// If you never want to read more than 4 byte use the CIA405.SDO_READ4 functionblock instead.
// Set xEnable to TRUE in online mode to get the program working.
PROGRAM SegmentedAndBlockReadExample
VAR
	xEnable       : BOOL; // Set this variable to true to start the example code.
	psData        : POINTER TO STRING(MAX_CHAR - 1) := ADR(aData); // Result: Device Name
	dwAbortCode	  : DWORD; //contains abort code in case of error

	SDORead    	  : CIA405.SDO_READ_DATA;
	RTrig 		  : Standard.R_TRIG;										  
	aData	      : ARRAY[0..MAX_CHAR] OF BYTE;
	udiDataLength : UDINT;
END_VAR
VAR CONSTANT
	MAX_CHAR : INT := 256;
END_VAR

RTrig(CLK := xEnable);

IF RTrig.Q THEN
	// Rising edge for xEnable detected ==> Prepare SDO write function block
	
	// ==> Initialize read buffer with 0 (clear old read results)
	MEMUtils.MemSet(pbyBuffer := ADR(aData[0]), byValue := 0, dwSize := SIZEOF(aData));
	
	// ==> Set udiDataLength to read buffer length.
	// Note: Do not forget setting udiDataLength each time when you start a new SDO read operation. 
	// This is necessary because udiDataLength is a VAR_IN_OUT variable and will be modified by SDORead function block!
	// It contains the number of valid bytes read by the function block.
	udiDataLength := SIZEOF(aData) - 1; //-1 only needed because CANopen strings are not null terminated! So we need one additional byte for the null termination. ==> Not needed for other datatypes!
END_IF

IF SDORead.CONFIRM THEN
	// SDO Read successful. aData contains data (= Device Name); udiDataLength contains number of bytes read (string length without null termination).
	xEnable := FALSE;
ELSIF SDORead.ERROR <> CiA405.CANOPEN_KERNEL_ERROR.CANOPEN_KERNEL_NO_ERROR THEN
	// Error occured
	IF SDORead.ERROR = CIA405.CANOPEN_KERNEL_ERROR.CANOPEN_KERNEL_OTHER_ERROR THEN
		//output error info contains abort code in little endian format
		MEMUtils.MemCpy(pbyDest := ADR(dwAbortCode), pbySrc := ADR(SDORead.ERRORINFO), dwSize := SIZEOF(dwAbortCode));
		MEMUtils.SwapLocalToIntel(pAddress := ADR(dwAbortCode), iSize := TO_INT(SIZEOF(dwAbortCode))); //function only swaps on big endian systems	
	END_IF
	xEnable := FALSE;
END_IF

SDORead(   Enable     := xEnable,
		   Network    := CANbus.NetId + 1, //CODESYS NetId starts by 0 (the number entered into the CANbus configurator); CiA405 NETWORK by 1; That is the reason why we have to increment it here.
           Timeout    := 0, //Timeout for SDO read in ms. Here: 0 ==> no timeout
           Device     := CANopenRemoteDevice.NodeID, // NodeID of destination device
           Channel    := 0, //SDO channel which should be used. 0 means auto channeling ==> the next free channel will be used. It depends on the slave which settings are working here but 0 and channel 1 is always working. 
           Index      := 16#1008, //object index which should be read ==> 16#1008sub0 = Device Name
           SubIndex   := 0, //object sub index which should be read ==> 16#1008sub0 = Device Name
		   MODE		  := CIA405.SDO_MODE.AUTO, //Use SDO mode AUTO ==> Mode will be selected automatically. Use SDO_MODE.BLOCK for forcing Block Transfer.
           Data       := ADR(aData), // Pointer to data buffer where result should be written to.
           DataLength := udiDataLength //VAR_IN: Length of data buffer; VAR_OUT: Length of data written to data buffer.
);

END_PROGRAM

// Device/Application/CANopen Master Examples/CiA405/SDO access/Block and Segmented/SegmentedAndBlockWriteExample
// This program uses CiA405.SDO_WRITE_DATA for writing more than 4 byte using segmented or block transfer.
//
// This example code writes a string into object 16#3000 of CANopenRemoteDevice.
// CiA405.SDO_WRITE_DATA is a universal function block which can be also used for expedited transfer (<= 4byte).
// If you never want to write more than 4 byte use the CIA405.SDO_WRITE4 functionblock instead.
// In online mode: Set psData to the string which should be written and then set xEnable to TRUE to get the program working.
// Afterwards you can check result in CANopenLocalDeviceExamples.strTestString. The Variable is mapped to object 16#3000 in object dictionary.
PROGRAM SegmentedAndBlockWriteExample
VAR
	xEnable       : BOOL; // Set this variable to true to start the example code.
	psData        : POINTER TO STRING(MAX_CHAR - 1) := ADR(aData); // String to write
	dwAbortCode	  : DWORD; //contains abort code in case of error

	SDOWrite      : CIA405.SDO_WRITE_DATA;							  
	aData	      : ARRAY[0..MAX_CHAR] OF BYTE;
END_VAR
VAR CONSTANT
	MAX_CHAR : INT := 256;
END_VAR

IF SDOWrite.CONFIRM THEN
	// SDO Write successful.
	xEnable := FALSE;
ELSIF SDOWrite.ERROR <> CiA405.CANOPEN_KERNEL_ERROR.CANOPEN_KERNEL_NO_ERROR THEN
	// Error occured
	IF SDOWrite.ERROR = CIA405.CANOPEN_KERNEL_ERROR.CANOPEN_KERNEL_OTHER_ERROR THEN
		//output error info contains abort code in little endian format
		MEMUtils.MemCpy(pbyDest := ADR(dwAbortCode), pbySrc := ADR(SDOWrite.ERRORINFO), dwSize := SIZEOF(dwAbortCode));
		MEMUtils.SwapLocalToIntel(pAddress := ADR(dwAbortCode), iSize := TO_INT(SIZEOF(dwAbortCode))); //function only swaps on big endian systems	
	END_IF
	xEnable := FALSE;
END_IF

SDOWrite(  Enable     := xEnable,
		   Network    := CANbus.NetId + 1, //CODESYS NetId starts by 0 (the number entered into the CANbus configurator); CiA405 NETWORK by 1; That is the reason why we have to increment it here.
           Timeout    := 0, //Timeout for SDO read in ms. Here: 0 ==> no timeout
           Device     := CANopenRemoteDevice.NodeID, // NodeID of destination device
           Channel    := 0, //SDO channel which should be used. 0 means auto channeling ==> the next free channel will be used. It depends on the slave which settings are working here but 0 and channel 1 is always working. 
           Index      := 16#3000, //object index which should be written ==> 16#3000 = simple string object
           SubIndex   := 0, //object sub index which should be written
		   MODE		  := CIA405.SDO_MODE.AUTO, //Use SDO mode AUTO ==> Mode will be selected automatically. Use SDO_MODE.BLOCK for forcing Block Transfer.
           Data       := ADR(aData), // Pointer to data buffer where result should be written to.
           DataLength := TO_UDINT(Stu.StrLenA(ADR(aData[0]))) //Length of data
);

END_PROGRAM

// Device/Application/CANopen Slave Examples/CANopenLocalDeviceExamples
PROGRAM CANopenLocalDeviceExamples
VAR
	// Variable strTestString is mapped to object 16#3000; It can be read and written by SDO.
	// Note: To avoid data inconsistencies the variable should be only accessed from bus cycle task!
	strTestString : STRING;
	
	xEventHandlerRegistered : BOOL;
	eventHandler : ObjectDictionaryEventHandler;
END_VAR

GetLocalDeviceInfoExample();
ChangeNodeIDExample();
NMTExample();

CountObjects();
GetPDOInfo();

ReadObjectExample1();
ReadObjectExample2();
WriteObjectExample1();
WriteObjectExample2();

IF NOT xEventHandlerRegistered THEN
	//Register object dictionary event handler
	xEventHandlerRegistered := CANopenLocalDevice.ObjectDictionary.RegisterCallback(eventHandler);
END_IF

END_PROGRAM

// Device/Application/CANopen Slave Examples/Diagnosis/GetLocalDeviceInfoExample
// This program shows how to get general slave information
FUNCTION GetLocalDeviceInfoExample : STRING
VAR_INPUT
END_VAR
VAR
	eSlaveState : _3SCSS.CANOPEN_STATE;
	usiNodeID : USINT;
END_VAR

// Get the CANopen state
eSlaveState := CANopenLocalDevice.State;
// Get the Node ID
usiNodeID := CANopenLocalDevice.NodeID;

END_FUNCTION

// Device/Application/CANopen Slave Examples/Network management/ChangeNodeIDExample
// This example changes the NodeID of the local device.
// Set xEnable to TRUE in online mode to get the program working.
PROGRAM ChangeNodeIDExample
VAR
	xEnable       : BOOL; // Set this variable to true to start the example code.
	usiNewNodeID  : USINT := 1; // Set the desired Node ID
	usiCurrentNodeID : USINT; // The current Node ID
	
	RTrig 	 : Standard.R_TRIG;
END_VAR

RTrig(CLK := xEnable);

IF RTrig.Q THEN
	CANopenLocalDevice.SetNodeID(usiNewNodeID);
	xEnable := FALSE;
END_IF

usiCurrentNodeID := CANopenLocalDevice.NodeID;

END_PROGRAM

// Device/Application/CANopen Slave Examples/Network management/NMTExample
// This program shows how to execute NMT commands on a local device.
// Note: The CANopenManager will automatically restart the slave if an unexpected state is detected.
// Set xEnable to TRUE in online mode to get the program working.
PROGRAM NMTExample
VAR
	xEnable       : BOOL; // Set this variable to true to start the example code.
	eNMTCommand	  : NMT_Command; // Set the desired NMT command
	eCurrentState : _3SCSS.CANOPEN_STATE; // The current slave state.
	RTrig 	 : Standard.R_TRIG;
END_VAR

RTrig(CLK := xEnable);

IF RTrig.Q THEN
	CASE eNMTCommand OF
		NMT_Command.PREOP:
			CANopenLocalDevice.SwitchToPreop();
		NMT_Command.RESET:
			CANopenLocalDevice.Reset();
		NMT_Command.START:
			CANopenLocalDevice.SwitchToOp();
		NMT_Command.STOP:
			CANopenLocalDevice.SwitchToStopped();
		NMT_Command.POWER_DOWN:
			CANopenLocalDevice.PowerDown(); //disables the slave
		NMT_Command.POWER_UP:
			CANopenLocalDevice.PowerUp(); //enables the slave
	END_CASE	

	xEnable := FALSE;
END_IF

eCurrentState := CANopenLocalDevice.State;

END_PROGRAM

// Device/Application/CANopen Slave Examples/Object Dictionary Access/Traverse object dictionary/CountObjects
// Following program shows how to iterate over all objects of the local object dictionary by using an ObjectIterator.
// It counts the number of objects and subobjects.
// Set xEnable to TRUE in online mode to get the program working.
PROGRAM CountObjects
VAR
	xEnable       : BOOL; // Set this variable to true to start the example code.
	udiObjectCount : UDINT; // Number of objects
	udiSubObjCount : UDINT; // Number of subobjects
	
	ObjIterator : _3SCSS.ObjectIterator;
	SubObjIterator : _3SCSS.SubObjectIterator;
	itfCurObj : _3SCSS.IODObject;
	itfCurSubObj : _3SCSS.IODSubObject;
	RTrig 	 : Standard.R_TRIG;
END_VAR

RTrig(CLK := xEnable);

IF RTrig.Q THEN
	udiObjectCount := 0;
	udiSubObjCount := 0;
	
	//Link Object Iterator to Object Dictionary
	ObjIterator.ObjectDictionary := CANopenLocalDevice.ObjectDictionary;
	
	//Go through all objects
	WHILE ObjIterator.MoveNext() DO
		itfCurObj := ObjIterator.Current; //Note: No NULL check necessary here because MoveNext returned TRUE.
		udiObjectCount := udiObjectCount + 1;
		
		//Link SubObjIterator with current Object
		SubObjIterator.Object := itfCurObj;
		
		//Go through all SubObjects
		WHILE SubObjIterator.MoveNext() DO
			itfCurSubObj := SubObjIterator.Current;
			udiSubObjCount := udiSubObjCount + 1;
		END_WHILE
	END_WHILE
	
	xEnable := FALSE;
END_IF

END_PROGRAM

// Device/Application/CANopen Slave Examples/Object Dictionary Access/Traverse object dictionary/GetPDOInfo
// Following program shows how to iterate over all objects of the local object dictionary by using an ObjectIterator.
// It creates a PDO statistic.
// Set xEnable to TRUE in online mode to get the program working.
PROGRAM GetPDOInfo
VAR
	xEnable       : BOOL; // Set this variable to true to start the example code.
	byTxPDOs : BYTE; // Number of transmit PDOs
	byActivatedTxPDOs : BYTE; // Number of activated transmit PDOs
	byRxPDOs : BYTE; // Number of receive PDOs
	byActivatedRxPDOs : BYTE; // Number of activated receive PDOs
	
	ObjIterator : _3SCSS.ObjectIterator;
	itfCurObj : _3SCSS.IODObject;
	itfCOBIDSubObj : _3SCSS.IODSubObject;
	pdwValue : POINTER TO DWORD;
	xPDOEnabled : BOOL;
	RTrig 	 : Standard.R_TRIG;
END_VAR

RTrig(CLK := xEnable);

IF RTrig.Q THEN
	byTxPDOs := 0;
	byActivatedTxPDOs := 0;
	byRxPDOs := 0;
	byActivatedRxPDOs := 0;
	
	//Link Object Iterator to Object Dictionary
	ObjIterator.ObjectDictionary := CANopenLocalDevice.ObjectDictionary;
	
	//Go through all objects
	WHILE ObjIterator.MoveNext() DO
		itfCurObj := ObjIterator.Current; //Note: No NULL check necessary here because MoveNext returned TRUE.
		IF itfCurObj.Index >= 16#1400 AND itfCurObj.Index <= 16#15FF THEN
			byRxPDOs := byRxPDOs + 1;
			//Check if PDO is enabled
			itfCOBIDSubObj := itfCurObj.GetSubObject(1);
			pdwValue := itfCOBIDSubObj.pData;
			_3SCSS.DecodePDOCOBID(dwValue := pdwValue^, xEnabled => xPDOEnabled);
			IF xPDOEnabled THEN
				byActivatedRxPDOs := byActivatedRxPDOs + 1;
			END_IF
		ELSIF itfCurObj.Index >= 16#1800 AND itfCurObj.Index <= 16#19FF THEN
			byTxPDOs := byTxPDOs + 1;
			//Check if PDO is enabled
			itfCOBIDSubObj := itfCurObj.GetSubObject(1);
			pdwValue := itfCOBIDSubObj.pData;
			_3SCSS.DecodePDOCOBID(dwValue := pdwValue^, xEnabled => xPDOEnabled);
			IF xPDOEnabled THEN
				byActivatedTxPDOs := byActivatedTxPDOs + 1;
			END_IF
		END_IF
	END_WHILE
	
	xEnable := FALSE;
END_IF

END_PROGRAM

// Device/Application/CANopen Slave Examples/Object Dictionary Access/Read Object/ReadObjectExample1
//This method is one possible implementation for reading an object (in this case the Identity Object 16#1018).
//This implementation reads the value by using the ReadObjectByAddress method.
// Set xEnable to TRUE in online mode to get the program working.
PROGRAM ReadObjectExample1
VAR
	xEnable       : BOOL; // Set this variable to true to start the example code.
	dwVendorID : DWORD; // VendorID read from local object dictionary
	dwProductCode : DWORD; // ProduceCode read from local object dictionary
	dwRevisionNumber : DWORD; // RevisionNumber read from local object dictionary
	xVendorIDAvailable : BOOL; // object dictionary contains object for VendorID 
	xProductCodeAvailable : BOOL; // object dictionary contains object for ProductCode 
	xRevisionNumberAvailable : BOOL; // object dictionary contains object for RevisionNumber 
	
	udiSize : UDINT;
	eAbortCode : _3SCSS.ABORT_CODE;
	RTrig 	 : Standard.R_TRIG;
END_VAR

RTrig(CLK := xEnable);

IF RTrig.Q THEN
	dwVendorID := 0;
	dwProductCode := 0;
	dwRevisionNumber := 0;
	xVendorIDAvailable := FALSE;
	xProductCodeAvailable := FALSE;
	xRevisionNumberAvailable := FALSE;
	
	//Reading Vendor ID
	//xCheckAccess = FALSE means that Access Rights should be ignored. Reading of a writeonly object will be possible.
	//xDataInBusOrder = FALSE means that data should be read in host byte order.
	udiSize := 4;
	eAbortCode := CANopenLocalDevice.ObjectDictionary.ReadObjectByAddress(wIndex := 16#1018, bySubIndex := 16#1, xCheckAccess := FALSE, xDataInBusOrder := FALSE, pbyData := ADR(dwVendorID), udiSize := udiSize);
	IF eAbortCode = _3SCSS.ABORT_CODE.SUCCESSFUL THEN
		xVendorIDAvailable := TRUE;
	END_IF
	
	//Reading Product Code
	udiSize := 4;
	eAbortCode := CANopenLocalDevice.ObjectDictionary.ReadObjectByAddress(wIndex := 16#1018, bySubIndex := 16#2, xCheckAccess := FALSE, xDataInBusOrder := FALSE, pbyData := ADR(dwProductCode), udiSize := udiSize);
	IF eAbortCode = _3SCSS.ABORT_CODE.SUCCESSFUL THEN
		xProductCodeAvailable := TRUE;
	END_IF
	
	//Reading Revision Number
	udiSize := 4;
	eAbortCode := CANopenLocalDevice.ObjectDictionary.ReadObjectByAddress(wIndex := 16#1018, bySubIndex := 16#3, xCheckAccess := FALSE, xDataInBusOrder := FALSE, pbyData := ADR(dwRevisionNumber), udiSize := udiSize);
	IF eAbortCode = _3SCSS.ABORT_CODE.SUCCESSFUL THEN
		xRevisionNumberAvailable := TRUE;
	END_IF
	
	xEnable := FALSE;
END_IF

END_PROGRAM

// Device/Application/CANopen Slave Examples/Object Dictionary Access/Read Object/ReadObjectExample2
//This method is one possible implementation for reading an object (in this case the Identity Object 16#1018).
//This implementation reads the value by using the ReadObject method.
// Set xEnable to TRUE in online mode to get the program working.
PROGRAM ReadObjectExample2
VAR
	xEnable       : BOOL; // Set this variable to true to start the example code.
	dwVendorID : DWORD; // VendorID read from local object dictionary
	dwProductCode : DWORD; // ProduceCode read from local object dictionary
	dwRevisionNumber : DWORD; // RevisionNumber read from local object dictionary
	xVendorIDAvailable : BOOL; // object dictionary contains object for VendorID 
	xProductCodeAvailable : BOOL; // object dictionary contains object for ProductCode 
	xRevisionNumberAvailable : BOOL; // object dictionary contains object for RevisionNumber 
	
	itfIdentityObject : _3SCSS.IODObject;
	udiSize : UDINT;
	eAbortCode : _3SCSS.ABORT_CODE;
	RTrig 	 : Standard.R_TRIG;
END_VAR

RTrig(CLK := xEnable);

IF RTrig.Q THEN
	dwVendorID := 0;
	dwProductCode := 0;
	dwRevisionNumber := 0;
	xVendorIDAvailable := FALSE;
	xProductCodeAvailable := FALSE;
	xRevisionNumberAvailable := FALSE;
	
	IF itfIdentityObject = 0 THEN
		itfIdentityObject := CANopenLocalDevice.ObjectDictionary.GetObject(16#1018);
	END_IF
	
	IF itfIdentityObject <> 0 THEN
		//Reading Vendor ID
		//xCheckAccess = FALSE means that Access Rights should be ignored. Reading of a writeonly object will be possible.
		//xDataInBusOrder = FALSE means that data should be read in host byte order.
		udiSize := 4;
		eAbortCode := CANopenLocalDevice.ObjectDictionary.ReadObject(itfObject := itfIdentityObject, bySubIndex := 16#1, xCheckAccess := FALSE, xDataInBusOrder := FALSE, pbyData := ADR(dwVendorID), udiSize := udiSize);
		IF eAbortCode = _3SCSS.ABORT_CODE.SUCCESSFUL THEN
			xVendorIDAvailable := TRUE;
		END_IF
		
		//Reading Product Code
		udiSize := 4;
		eAbortCode := CANopenLocalDevice.ObjectDictionary.ReadObject(itfObject := itfIdentityObject, bySubIndex := 16#2, xCheckAccess := FALSE, xDataInBusOrder := FALSE, pbyData := ADR(dwProductCode), udiSize := udiSize);
		IF eAbortCode = _3SCSS.ABORT_CODE.SUCCESSFUL THEN
			xProductCodeAvailable := TRUE;
		END_IF
		
		//Reading Revision Number
		udiSize := 4;
		eAbortCode := CANopenLocalDevice.ObjectDictionary.ReadObject(itfObject := itfIdentityObject, bySubIndex := 16#3, xCheckAccess := FALSE, xDataInBusOrder := FALSE, pbyData := ADR(dwRevisionNumber), udiSize := udiSize);
		IF eAbortCode = _3SCSS.ABORT_CODE.SUCCESSFUL THEN
			xRevisionNumberAvailable := TRUE;
		END_IF
	END_IF
	
	xEnable := FALSE;
END_IF

END_PROGRAM

// Device/Application/CANopen Slave Examples/Object Dictionary Access/Write Object/WriteObjectExample1
// This method is one possible implementation for writing an object value (in this case SYNC COBID 16#1005).
// Set xEnable to TRUE in online mode to get the program working.
PROGRAM WriteObjectExample1
VAR
	xEnable       : BOOL; // Set this variable to true to start the example code.
	dwSyncCOBID : DWORD := 16#80; // SyncCOBID which should be written to local object dictionary
	xWriteSuccessful : BOOL;
	
	udiSize : UDINT;
	eAbortCode : _3SCSS.ABORT_CODE;
	RTrig 	 : Standard.R_TRIG;
END_VAR

RTrig(CLK := xEnable);

IF RTrig.Q THEN
	udiSize := SIZEOF(dwSyncCOBID);
	eAbortCode := CANopenLocalDevice.ObjectDictionary.WriteObjectByAddress(wIndex := 16#1005, bySubIndex := 0, xCheckAccess := TRUE, xDataInBusOrder := FALSE, pbyData := ADR(dwSyncCOBID), udiSize := udiSize);
	xWriteSuccessful := eAbortCode = _3SCSS.ABORT_CODE.SUCCESSFUL;
	xEnable := FALSE;
END_IF

END_PROGRAM

// Device/Application/CANopen Slave Examples/Object Dictionary Access/Write Object/WriteObjectExample2
// This method is one possible implementation for writing an object value (in this case SYNC COBID 16#1005).
// Set xEnable to TRUE in online mode to get the program working.
PROGRAM WriteObjectExample2
VAR
	xEnable       : BOOL; // Set this variable to true to start the example code.
	dwSyncCOBID : DWORD := 16#80; // SyncCOBID which should be written to local object dictionary
	xWriteSuccessful : BOOL;
	
	itfSyncCOBID : _3SCSS.IODObject;
	udiSize : UDINT;
	eAbortCode : _3SCSS.ABORT_CODE;
	RTrig 	 : Standard.R_TRIG;
END_VAR

RTrig(CLK := xEnable);

IF RTrig.Q THEN
	xWriteSuccessful := FALSE;
	IF itfSyncCOBID = 0 THEN
		itfSyncCOBID := CANopenLocalDevice.ObjectDictionary.GetObject(wIndex := 16#1005);
	END_IF
	
	IF itfSyncCOBID <> 0 THEN
		udiSize := SIZEOF(dwSyncCOBID);
		//xCheckAccess = TRUE means that AccessType should be checked. Writing on a readonly object will fail in this case. By setting xCheckAccess to false writing on a readonly object is possible.
		//xDataInBusOrder = FALSE means that data is in host byte order.
		eAbortCode := CANopenLocalDevice.ObjectDictionary.WriteObject(itfObject := itfSyncCOBID, bySubIndex := 0, xCheckAccess := TRUE, xDataInBusOrder := FALSE, pbyData := ADR(dwSyncCOBID), udiSize := udiSize);
		xWriteSuccessful := eAbortCode = _3SCSS.ABORT_CODE.SUCCESSFUL;
	END_IF
	xEnable := FALSE;
END_IF

END_PROGRAM

// Device/Application/CANopen Slave Examples/Object Dictionary Access/Event Handler/ObjectDictionaryEventHandler
// This function block implement an Object Dictionary event handler.
// Object Dictionary event handlers will be informed every time an object will be read or written.
// The event handler has the possibility to abort a pending read or write request with an appropriate abort code.
// The evemt handler is instantiated and registered in CANopenLocalDeviceExample PRG.
FUNCTION_BLOCK ObjectDictionaryEventHandler IMPLEMENTS _3SCSS.IODCallback
VAR_INPUT
END_VAR
VAR_OUTPUT
END_VAR
VAR
END_VAR

METHOD OnObjectChanged
VAR_INPUT
	(*Corresponding object*)
	itfObject	: _3SCSS.IODObject;
	(*Corresponding subobject*)
	itfSubObject	: _3SCSS.IODSubObject;
END_VAR
VAR
	strLogMsg : STRING;
END_VAR
// This method will be called by the CANopen Slave stack if an object value has changed.

// Just add a log message to the PLC logger
strLogMsg := 'CANopenLocalDevice: Object value changed 16#';
strLogMsg := Standard.CONCAT(strLogMsg, TO_HEXSTRING(itfObject.Index));
strLogMsg := Standard.CONCAT(strLogMsg, 'sub');
strLogMsg := Standard.CONCAT(strLogMsg, TO_HEXSTRING(itfSubobject.SubIndex));
CmpLog.LogAdd2(CmpLog.LOG_STD_LOGGER, 0, CmpLog.LogClass.LOG_INFO, 0, 0, strLogMsg);
END_METHOD

METHOD OnReadObject : _3SCSS.ABORT_CODE
VAR_INPUT
	(*Object to be read*)
	itfObject	: _3SCSS.IODObject;
	(*Subobject to be read*)
	itfSubObject	: _3SCSS.IODSubObject;
END_VAR
VAR
	strLogMsg : STRING;
END_VAR
// This method will be called by the CANopen Slave stack when a SDO read request is pending. You can return an appropriate abort code if read request should be aborted by SDO server.

// Just add a log message to the PLC logger
strLogMsg := 'CANopenLocalDevice: Read attempt on object 16#';
strLogMsg := Standard.CONCAT(strLogMsg, TO_HEXSTRING(itfObject.Index));
strLogMsg := Standard.CONCAT(strLogMsg, 'sub');
strLogMsg := Standard.CONCAT(strLogMsg, TO_HEXSTRING(itfSubobject.SubIndex));
CmpLog.LogAdd2(CmpLog.LOG_STD_LOGGER, 0, CmpLog.LogClass.LOG_INFO, 0, 0, strLogMsg);

OnReadObject := _3SCSS.ABORT_CODE.SUCCESSFUL; //If read operation should be aborted you can return an appropriate abort code here.
END_METHOD

METHOD OnWriteObject : _3SCSS.ABORT_CODE
VAR_INPUT
	itfObject	: _3SCSS.IODObject;
	itfSubObject	: _3SCSS.IODSubObject;
	pbyData	: POINTER TO BYTE;
	udiSize	: UDINT;
END_VAR
VAR
	strLogMsg : STRING;
END_VAR
// This method will be called by the CANopen Slave stack when a SDO write request is pending. You can return an appropriate abort code if write request should be aborted by SDO server.
// If an abort code will be returned object value remains unchanged.

// Just add a log message to the PLC logger
strLogMsg := 'CANopenLocalDevice: Write attempt on object 16#';
strLogMsg := Standard.CONCAT(strLogMsg, TO_HEXSTRING(itfObject.Index));
strLogMsg := Standard.CONCAT(strLogMsg, 'sub');
strLogMsg := Standard.CONCAT(strLogMsg, TO_HEXSTRING(itfSubobject.SubIndex));
CmpLog.LogAdd2(CmpLog.LOG_STD_LOGGER, 0, CmpLog.LogClass.LOG_INFO, 0, 0, strLogMsg);

OnWriteObject := _3SCSS.ABORT_CODE.SUCCESSFUL; //If write operation should be aborted you can return an appropriate abort code here.
END_METHOD

END_FUNCTION_BLOCK

// Device/Application/CANopen Slave Examples/Object Dictionary Access/Event Handler/TO_HEXSTRING
FUNCTION TO_HEXSTRING : STRING(8)
VAR_INPUT
	value : UDINT;
END_VAR
VAR
	i : DINT;
	nibbleValue : UDINT;
	txt : POINTER TO BYTE;
	hex : POINTER TO BYTE;
	hexTable : STRING(17) := '0123456789ABCDEF ';
	pos : UDINT := 7;
	udiBitLength : UDINT;
	udiStringLength : UDINT;
END_VAR

txt := ADR(TO_HEXSTRING);
hex := ADR(hexTable);

IF value <> 0 THEN
	udiBitLength := TO_UDINT(LOG(value) / LOG(2)) + 1;
ELSE
	udiBitLength := 8;
END_IF

udiStringLength := ((udiBitLength + 7) / 8) * 2;
IF udiStringLength <= 8 THEN
	pos := udiStringLength - 1;
	
	FOR i := 0 TO TO_DINT(udiStringLength - 1) DO
		nibbleValue := SHR(value, 4 * i) AND 16#F;
		txt[pos] := hex[nibbleValue];
		pos := pos - 1;
	END_FOR
	
	txt[udiStringLength] := 0;
END_IF

END_FUNCTION

// Device/Application/CANopen Master Examples/CiA405/Network management/NMT_Example
// The following program sends a NMT command to the CANopenRemoteDevice attached below the CANopen_Manager.
// Set eState to the desired NMT command and xEnable to TRUE in online mode to get the program working.
PROGRAM NMT_Example
VAR
	xEnable : BOOL; // Set this variable to true to start the example code. Variable will be set to FALSE if NMT finished execution.
	eState : CIA405.TRANSITION_STATE := CIA405.TRANSITION_STATE.RESET_NODE; // NMT command which should be sent.
	
	NMT : CIA405.NMT;
END_VAR

IF NMT.CONFIRM = TRUE THEN
	// NMT command successful.
	xEnable := FALSE;
ELSIF NMT.ERROR <> CIA405.CANOPEN_KERNEL_ERROR.CANOPEN_KERNEL_NO_ERROR THEN
	// an error occured while processing NMT e.g. wrong NodeID or NetworkID
	xEnable := FALSE;
END_IF

NMT(	ENABLE := xEnable,
		NETWORK := CANbus.NetId + 1, //CODESYS NetId starts by 0 (the number entered into the CANbus configurator); CiA405 NETWORK by 1; That is the reason why we have to increment it here.
		TIMEOUT := 0, // no timeout for GetState needed because it is processed locally.
		DEVICE := CANopenRemoteDevice.NodeID, // Use 0 if you want to send a NMT all command!
		STATE := eState //the NMT command which should be sent
);

END_PROGRAM

// Device/Application/CANopen Master Examples/CiA405/Network management/GetCANopenManagerNodeIDExample
// This program reads the NodeID of the local CANopenManager.
// Set xEnable to TRUE in online mode to get the program working.
PROGRAM GetCANopenManagerNodeIDExample
VAR
	xEnable : BOOL; // Set this variable to true to start the example code. Variable will be set to FALSE if GetNodeID finished execution.
	NodeID : CiA405.DEVICE; // Result: CANopen NodeID
	
	GetNodeID : CIA405.GET_LOCAL_NODE_ID;
END_VAR

IF GetNodeID.CONFIRM = TRUE THEN
	// GetNodeID successful. Output device contains CANopenManager NodeID.
	NodeID := GetNodeID.DEVICE;
	xEnable := FALSE;
ELSIF GetNodeID.ERROR <> CIA405.CANOPEN_KERNEL_ERROR.CANOPEN_KERNEL_NO_ERROR THEN
	// an error occured while processing GetState e.g. wrong NodeID or NetworkID
	xEnable := FALSE;
END_IF

GetNodeID( 	ENABLE := xEnable,
		  	NETWORK := CANbus.NetId + 1, //CODESYS NetId starts by 0 (the number entered into the CANbus configurator); CiA405 NETWORK by 1; That is the reason why we have to increment it here.
		  	TIMEOUT := 0 // no timeout for GetNodeID needed because it is processed locally.
);

END_PROGRAM

// Device/Application/CANopen Master Examples/Stack API/CANopenManagerAPI
// This example program shows how to use the CANopen Manager API.
PROGRAM CANopenManagerAPI
VAR
	pDevice : POINTER TO _3SCOS.CANRemoteDevice;
	kernelState : _3SCOS.CANOPEN_KERNEL_STATE;
	xAllMandatorySlaveBooted : BOOL;
	xAllOptionalSlavesBooted : BOOL;
	wNMTInhibitTime : WORD;
	
	udiNumberOfSlaves : UDINT; //How many slaves are attached below the CANopenManager
	udiNumberOfOperationalSlaves : UDINT; //How many slaves are in OPERATIONAL
	udiTotalConfigurationErrors : UDINT; //How many configuration errors (= SDO aborts) happened in configuration phase?
	udiNumberOfSlavesWithActivatedErrorControl : UDINT; //How many slaves have Error control (= Heartbeat or Nodeguarding) activated?
	
	usiCurrentNodeID : USINT;
	
	xEventHandlerRegistered : BOOL;
	EventHandler : CANopenManagerEventHandler; // CANopenManager event handler instance
END_VAR

//gets the CANopenManager kernel state ==> see also CiA405.GET_CANOPEN_KERNEL_STATE
kernelState := CANopen_Manager.KernelState;

//Are all mandatory slaves found and configured by CANopenManager?
xAllMandatorySlaveBooted := CANopen_Manager.MandatorySlavesBooted;

//Are all optional slaves found and configured by CANopenManager?
xAllOptionalSlavesBooted := CANopen_Manager.OptionalSlavesBooted;

//Gets or sets the NMT Inhibit Time (unit: multiple of 100us).
wNMTInhibitTime := CANopen_Manager.NMTInhibitTime;

//go through all remote devices of CANopen_Manager and collect some statistics
udiNumberOfSlaves := 0;
udiNumberOfOperationalSlaves := 0;
udiTotalConfigurationErrors := 0;
udiNumberOfSlavesWithActivatedErrorControl := 0;

FOR usiCurrentNodeID := 1 TO 127 DO
	pDevice := CANopen_Manager.GetSlaveByNodeID(usiCurrentNodeID);
	IF pDevice <> 0 THEN
		//count slaves
		udiNumberOfSlaves := udiNumberOfSlaves + 1;
		
		//Get the slave state ==> see also CiA405.GET_STATE
		IF pDevice^.CANopenState = _3SCOS.DEVICE_STATE.OPERATIONAL THEN
			udiNumberOfOperationalSlaves := udiNumberOfOperationalSlaves + 1;
		END_IF
		
		//Sum up configuration errors. 
		//NOTE: For getting more detailed information you can add the Compiler Define CANOPEN_DEBUG to the application.
		//Then perform a new download and go to the PLC logger. It contains further information for debugging purpose. 
		udiTotalConfigurationErrors := udiTotalConfigurationErrors + pDevice^.ConfigurationErrors;
		
		//Sum up all slaves with error control activated
		IF pDevice^.ErrorControlActivated THEN
			udiNumberOfSlavesWithActivatedErrorControl := udiNumberOfSlavesWithActivatedErrorControl + 1;
		END_IF
	END_IF
END_FOR

// Register a CANopen Manager event handler: An event handler can be used to add additional code to the stack state machine.
// In this example a SDO Read for CANopenRemoteDevice is performed after SDO configuration phase.
// For further details see CANopenManagerEventHandler.EventCallback
IF NOT xEventHandlerRegistered THEN
	xEventHandlerRegistered := CANopen_Manager.RegisterEventHandler(EventHandler);
END_IF

END_PROGRAM

// Device/Application/CANopen Master Examples/Stack API/Events/CANopenManagerEventHandler
// The following function block shows how to implement a CANopenEventHandler which could be registered
// at CANopen_Manager function block instance (see PRG CANopenManagerAPI).
// See EventCallback method for more details.
FUNCTION_BLOCK CANopenManagerEventHandler IMPLEMENTS _3SCOS.ICANopenEventHandler //Interface needed for registering at CANopen_Manager instance.
VAR_INPUT
END_VAR
VAR_OUTPUT
END_VAR
VAR
	read: CIA405.SDO_READ4; // used to read the device type
	dwDeviceTypeRead : DWORD; // device type read from CANopenRemoteDevice
	xDeviceTypeValid : BOOL; // device type read successfully
END_VAR

// Nothing to do!

// This method implements a CANopen Manager event handler.
// Every time the SDO configuration phase for CANopenRemoteDevice has finished, the Device Type will be read by this handler.
// As long as Event Handler returns FALSE the state machine of CANopenRemoteDevice is stopped. 
METHOD EventCallback : BOOL
VAR_INPUT
	(*Event Type*)
	eEvent	: _3SCOS.CANopenEvent;
	(*NodeID associated with the event; 0 if not relevant.*)
	usiNodeID	: USINT;
END_VAR
CASE eEvent OF
	_3SCOS.CANopenEvent.AFTER_SDO_CONFIG:
		IF usiNodeID = CANopenRemoteDevice.NodeID THEN
			//Read Device Type of slave
			read(ENABLE := TRUE, NETWORK := CANbus.NetId + 1, DEVICE := usiNodeID, CHANNEL := 0, INDEX := 16#1000, SUBINDEX := 16#0);
			IF read.CONFIRM OR read.ERROR <> CIA405.CANOPEN_KERNEL_ERROR.CANOPEN_KERNEL_NO_ERROR THEN
				IF read.CONFIRM THEN
					//value was read without error
					// ==> Copy data from SDO read function block
					MEMUtils.MemCpy(pbyDest := ADR(dwDeviceTypeRead), pbySrc := ADR(read.DATA[1]), dwSize := SIZEOF(dwDeviceTypeRead));
					//==> On big endian systems: dwValue has to be swapped to CANopen byte order (= Little Endian).
					MEMUtils.SwapLocalToIntel(pAddress := ADR(dwDeviceTypeRead), iSize := TO_INT(SIZEOF(dwDeviceTypeRead))); //function only swaps on big endian systems
					xDeviceTypeValid := TRUE;
				ELSE
					xDeviceTypeValid := FALSE;
				END_IF
				
				read(ENABLE := FALSE);
				EventCallback := TRUE; //Event handled ==> resume state machine of CANopenRemoteDevice
			END_IF
		ELSE
			EventCallback := TRUE; // no specific handling for other nodes
		END_IF
	ELSE
		EventCallback := TRUE; // no specific handling for other events
END_CASE
END_METHOD

END_FUNCTION_BLOCK

// Device/Application/CANopen Master Examples/Stack API/CANopenRemoteDeviceAPI
// This example program shows how to use the CANopen Remotedevice API.
PROGRAM CANopenRemoteDeviceAPI
VAR
	slaveState : _3SCOS.DEVICE_STATE;
	uiConfigurationErrors : UINT;
	xErrorControlActivated : BOOL;
	pCANopenManager : POINTER TO _3SCOS.CANopenManager;
END_VAR

//Gets the pointer to the CANopenManager
pCANopenManager := CANopenRemoteDevice.pCANopenManager;

//Set Bootup Timeout of slave to 10 seconds
CANopenRemoteDevice.BootupTimeout := 10000000; // unit: us
		
//Get the slave state ==> see also CiA405.GET_STATE
slaveState := CANopenRemoteDevice.CANopenState;

//How many configuration errors (= SDO aborts) happened in configuration phase of the slave?
uiConfigurationErrors := CANopenRemoteDevice.ConfigurationErrors;

//Error control (= Heartbeat or Nodeguarding) for slave activated?
xErrorControlActivated := CANopenRemoteDevice.ErrorControlActivated;

//Set the NMT Error behaviour of slave to RESTART_SLAVE.
//This means: If a Heartbeat or Nodeguarding error is detected for the slave it will be automatically restarted (=default behaviour).
CANopenRemoteDevice.NMTErrorBehaviour := _3SCOS.NMT_ERROR_BEHAVIOUR.RESTART_SLAVE;

END_PROGRAM

// Device/Application/CANbus Examples/CANbusExamples
PROGRAM CANbusExamples
VAR
END_VAR

ChangeBaudrate(); // How to change the baudrate of a CANbus
EnableDisableCANbus(); // How to enable/disable a CANbus

END_PROGRAM

// Device/Application/CANbus Examples/Change CANbus settings (Reconfigure)/ChangeBaudrate
// This program shows how to change the baudrate of a CANbus by using CAA Device Diagnosis Reconfigure.
// Make sure that PLC setting "Enable Diagnosis for devices" is activated!
// Set xEnable to TRUE in online mode to get the program working.
PROGRAM ChangeBaudrate
VAR
	xEnable       : BOOL; // Set this variable to true to start the example code.
	usiNetID	  : USINT; // NetID of CANbus on which baudrate change should be performed
	wBaudrate : WORD := 1000; // Set new Baudrate 
	
	iState : INT := 0;
	pCANBus : POINTER TO CANbusDevice.CANbus_Diag;
	reconfigure : DED.Reconfigure;
	RTrig 	 : Standard.R_TRIG;
END_VAR

CASE iState OF
	0:
		//Detect rising edge
		RTrig(CLK := xEnable);
		IF RTrig.Q THEN
			iState := 1;
		END_IF	

	1: 
		// Get the CANbus instance for a specific Network ID
		pCANBus := GetCANbus(usiNetID); // Here the pointer to the CANbus instance with NetID = usiNetID is calculated (the generic way!), 
									    // but you can also use the CANbus FB instance directly. For example: CANbus_1.SetBaudrate(wBaudrate)
		IF pCANBus <> 0 THEN
			// CANbus found ==> Set new Baudrate. Note: Baudrate change takes effect after reconfigure.
			// It is also possible changing NetID by calling SetNetID.
			pCANBus^.SetBaudrate(wBaudrate);
			iState := 2;
		ELSE
			// Error : No CANbus found
			iState := 3;
		END_IF
		
	2:
		// perform reconfigure
		reconfigure(xExecute := TRUE, itfNode := pCANBus^); // Here we use the pointer to the CANbus and dereference it. 
															// So we get the INode interface which is implemented by this instance (==> the generic way). 
															// But you can also use the CANbus FB instance directly. For Example: reconfigure(xExecute := TRUE, itfNode := CANbus_1)
		
		IF reconfigure.xDone OR reconfigure.xError THEN 	// Note: Add error handling for xError!
			reconfigure(xExecute := FALSE);
			iState := 3;
		END_IF
		
	3:
		iState := 0;
		xEnable := FALSE;
END_CASE

END_PROGRAM

// Device/Application/CANbus Examples/Query CANbus/GetCANbus
// Gets the pointer to the CANbus device instance by using CAA Device Diagnosis and __QUERYPOINTER.
// Make sure that PLC setting "Enable Diagnosis for devices" is activated!
FUNCTION GetCANbus : POINTER TO CANbusDevice.CANbus_Diag
VAR_INPUT
	usiNetID : USINT; // Network ID of CANbus
END_VAR
VAR
	itfNode : DED.INode;
	itfBus : DED.IBus;
	buiBusInfo : DED.BUS_INFO;
END_VAR

// first get PLC device
itfNode := DED.GetRoot();

// Go through device tree and search for CANbus
WHILE itfNode <> 0 DO
	itfBus := DED.INode_TO_IBus(itfNode); // check if current node is a bus
	IF itfBus <> 0 THEN
		// current node is a bus
		IF itfBus.GetBusInfo(buiBusInfo) = DED.ERROR.NO_ERROR THEN // get bus information
			IF buiBusInfo.eType = DED.BUS_TYPE.CAN AND_THEN buiBusInfo.idSystem = usiNetID THEN //check if it is a CANbus and compare NetID
				// CANbus found!
				__QUERYPOINTER(itfBus, GetCANbus); // Get CANbus_Diag instance pointer
				EXIT; // finished!
			END_IF
		END_IF
	END_IF
	
	itfBus := 0;
	itfNode := DED.GetNextNode(itfNode); // traverse tree ==> go to next node
END_WHILE

END_FUNCTION

// Device/Application/CANbus Examples/Change CANbus settings (Reconfigure)/EnableDisableCANbus
// This program shows how to enable/disable a complete CANbus by using CAA Device Diagnosis Reconfigure.
// This example project is not only appliable on CANbus nodes. It works also on all other nodes (e.g. CANopen Manager, CANopen Local Device, ...).
// Make sure that PLC setting "Enable Diagnosis for devices" is activated!
// Set xEnable to TRUE in online mode to get the program working.
PROGRAM EnableDisableCANbus
VAR
	xEnable       : BOOL; // Set this variable to true to start the example code.
	usiNetID	  : USINT; // NetID of CANbus which should be enabled/disabled
	xEnableCANbus : BOOL; // TRUE: Enable CANbus, FALSE: Disable CANbus
	
	iState : INT := 0;
	
	pCANbus : POINTER TO CANbusDevice.CANbus_Diag;
	reconfigure : DED.Reconfigure;
	RTrig 	 : Standard.R_TRIG;
END_VAR

CASE iState OF
	0:
		//Detect rising edge
		RTrig(CLK := xEnable);
		IF RTrig.Q THEN
			iState := 1;
		END_IF
	1:
		// Get the CANbus instance for a specific Network ID
		pCANbus := GetCANbus(usiNetID);
		
		IF pCANbus <> 0 THEN
			// CANbus found ==> Set enable flag. Note: Enable flag takes effect after reconfigure.
			pCANbus^.Enable := xEnableCANbus;
			iState := 2;
		ELSE
			// Error : No CANbus found
			iState := 3;
		END_IF
		
	2:
		// perform reconfigure
		reconfigure(xExecute := TRUE, itfNode := pCANbus^); // Here we use the pointer to the CANbus and dereference it.
															// So we get the INode interface which is implemented by this instance (==> the generic way). 
															// But you can also use the CANbus FB instance directly. For Example: reconfigure(xExecute := TRUE, itfNode := CANbus_1)

		IF reconfigure.xDone OR reconfigure.xError THEN     // Note: Add error handling for xError!
			reconfigure(xExecute := FALSE);
			iState := 3;
		END_IF
		
	3:
		iState := 0;
		xEnable := FALSE;
END_CASE

END_PROGRAM
